KUKA KRL program: ap_2.src, ap_2.dat

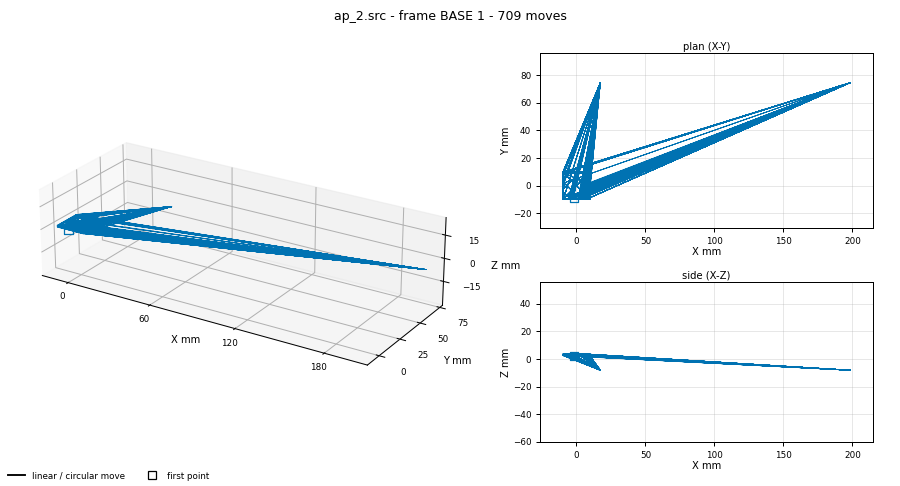
[picture p0: tool path of ap_2.src in frame BASE 1, 709 of 709 moves have a stored position in this frame; points joined in program order, loops and branches not executed]
--- ap_2.src ---
&ACCESS RVP
&REL 65
&PARAM DISKPATH = KRC:\R1\Program
DEF ap_2 ( )
   ;FOLD INI;%{PE}
     ;FOLD BASISTECH INI
       GLOBAL INTERRUPT DECL 3 WHEN $STOPMESS==TRUE DO IR_STOPM ( )
       INTERRUPT ON 3
       BAS (#INITMOV,0 )
     ;ENDFOLD (BASISTECH INI)
     ;FOLD USER INI
       ;Make your modifications here
     ;ENDFOLD (USER INI)
   ;ENDFOLD (INI)

   BAS (#VEL_PTP, 0020.0000)
   BAS (#ACC_PTP, 0020.0000)

   ;-----SET LIN AND ARC MOTION VARIABLES-----
   $VEL.ORI1 = 0350.0000
   $VEL.ORI2 = 0350.0000

   $ACC.CP = 0005.0000
   $ACC.ORI1 = 1000.0000
   $ACC.ORI2 = 1000.0000

   ;-----APPROXIMATION-----
   $APO.CVEL = 0100
   $APO.CPTP = 0100
   $APO.CDIS = 0006.0000
   $APO.CORI = 0090.0000

   BAS (#BASE, 1) ;Positioner
   BAS (#TOOL, 1) ;Vrashatel

   BAS(#VEL_PTP,15)                         ;;Set PTP Axis Velocity
   BAS(#ACC_PTP,50)                         ;;Set PTP Axis Acceleration
   PTP{A1 -92,A2 -133,A3 132,A4 7,A5 50,A6 -10}
   $VEL.CP = 0.060
   LIN  {X -1.968, Y -9.039, Z 2.300, A 0.000, B 0.000, C 0.000} C_DIS
   $VEL.CP = 0.060
   LIN  {X -5.102, Y -9.039, Z 2.300, A 0.000, B 0.000, C 0.000} C_DIS
   $VEL.CP = 0.060
   LIN  {X -9.039, Y -5.102, Z 2.300, A 0.000, B 0.000, C 0.000} C_DIS
   $VEL.CP = 0.060
   LIN  {X -9.039, Y -9.039, Z 2.300, A 0.000, B 0.000, C 0.000} C_DIS
   $VEL.CP = 0.060
   LIN  {X 9.039, Y 9.039, Z 2.300, A 0.000, B 0.000, C 0.000} C_DIS
   $VEL.CP = 0.060
   LIN  {X 9.040, Y 9.040, Z 2.300, A 0.000, B 0.000, C 0.000} C_DIS
   $VEL.CP = 0.060
   LIN  {X 9.039, Y 5.102, Z 2.300, A 0.000, B 0.000, C 0.000} C_DIS
   $VEL.CP = 0.060
   LIN  {X 5.102, Y 9.039, Z 2.300, A 0.000, B 0.000, C 0.000} C_DIS
   $VEL.CP = 0.060
   LIN  {X 1.968, Y 9.039, Z 2.300, A 0.000, B 0.000, C 0.000} C_DIS
   $VEL.CP = 0.060
   LIN  {X -9.039, Y -1.968, Z 2.300, A 0.000, B 0.000, C 0.000} C_DIS
   $VEL.CP = 0.060
   LIN  {X -9.039, Y 1.968, Z 2.300, A 0.000, B 0.000, C 0.000} C_DIS
   $VEL.CP = 0.060
   LIN  {X 1.968, Y -9.039, Z 2.300, A 0.000, B 0.000, C 0.000} C_DIS
   $VEL.CP = 0.060
   LIN  {X 9.040, Y -9.040, Z 2.300, A 0.000, B 0.000, C 0.000} C_DIS

;FOLD ARCOFF WDAT2 LIN P4 CPDAT2 Tool[1]:cmttorch Base[1]:vrashatel ;%{PE}
  ;FOLD Parameters ;%{h}
    ;Params IlfProvider=kukaroboter.arctech.arcofflin; Kuka.IsGlobalPoint=False; Kuka.PointName=P4; Kuka.BlendingEnabled=False; Kuka.MoveDataName=CPDAT2; Kuka.VelocityPath=0.01; Kuka.CurrentCDSetIndex=0; Kuka.MovementParameterFieldEnabled=True; ArcTech.WdatVarName=WDAT2; ArcTech.Basic=3.4.3.1264
  ;ENDFOLD
  $BWDSTART = FALSE
  LDAT_ACT = LCPDAT2
  FDAT_ACT = FP4
  BAS(#CP_PARAMS, gArcBasVelDefinition)
  SET_CD_PARAMS (0)
  TRIGGER WHEN PATH = ArcGetPath(#ArcOffBefore, WDAT2) DELAY = 0 DO ArcMainNG(#ArcOffBeforeOffStd, WDAT2, WP4) PRIO = -1
  TRIGGER WHEN PATH = ArcGetPath(#OnTheFlyArcOff, WDAT2) DELAY = 0 DO ArcMainNG(#ArcOffMoveStd, WDAT2, WP4) PRIO = -1
  ArcMainNG(#ArcOffBeforeMoveStd, WDAT2, WP4)
  LIN XP4
  ArcMainNG(#ArcOffAfterMoveStd, WDAT2, WP4)
;ENDFOLD
   $VEL.CP = 0.080
   LIN  {X 9.039, Y -9.039, Z 2.300, A 0.000, B 0.000, C 0.000} C_DIS

;FOLD ARCON WDAT1 LIN P3 Vel=0.5 m/s CPDAT1 Tool[1]:cmttorch Base[1]:vrashatel ;%{PE}
  ;FOLD Parameters ;%{h}
    ;Params IlfProvider=kukaroboter.arctech.arconlin; Kuka.IsGlobalPoint=False; Kuka.PointName=P3; Kuka.BlendingEnabled=False; Kuka.MoveDataName=CPDAT1; Kuka.VelocityPath=0.5; Kuka.CurrentCDSetIndex=0; Kuka.MovementParameterFieldEnabled=True; ArcTech.WdatVarName=WDAT1; ArcTech.Basic=3.4.3.1264
  ;ENDFOLD
  $BWDSTART = FALSE
  LDAT_ACT = LCPDAT1
  FDAT_ACT = FP3
  BAS(#CP_PARAMS, 0.5)
  SET_CD_PARAMS (0)
  TRIGGER WHEN DISTANCE = 1 DELAY = ArcGetDelay(#PreDefinition, WDAT1) DO ArcMainNG(#PreDefinition, WDAT1, WP3) PRIO = -1
  TRIGGER WHEN PATH = ArcGetPath(#OnTheFlyArcOn, WDAT1) DELAY = ArcGetDelay(#GasPreflow, WDAT1) DO ArcMainNG(#GasPreflow, WDAT1, WP3) PRIO = -1
  TRIGGER WHEN PATH = ArcGetPath(#OnTheFlyArcOn, WDAT1) DELAY = 0 DO ArcMainNG(#ArcOnMoveStd, WDAT1, WP3) PRIO = -1
  ArcMainNG(#ArcOnBeforeMoveStd, WDAT1, WP3)
  LIN XP3
  ArcMainNG(#ArcOnAfterMoveStd, WDAT1, WP3)
;ENDFOLD
   $VEL.CP = 0.060
   LIN  {X -9.039, Y 9.039, Z 2.300, A 0.000, B 0.000, C 0.000} C_DIS
   $VEL.CP = 0.060
   LIN  {X -9.040, Y 9.040, Z 2.300, A 0.000, B 0.000, C 0.000} C_DIS

;FOLD ARCOFF WDAT2 LIN P4 CPDAT2 Tool[1]:cmttorch Base[1]:vrashatel ;%{PE}
  ;FOLD Parameters ;%{h}
    ;Params IlfProvider=kukaroboter.arctech.arcofflin; Kuka.IsGlobalPoint=False; Kuka.PointName=P4; Kuka.BlendingEnabled=False; Kuka.MoveDataName=CPDAT2; Kuka.VelocityPath=0.01; Kuka.CurrentCDSetIndex=0; Kuka.MovementParameterFieldEnabled=True; ArcTech.WdatVarName=WDAT2; ArcTech.Basic=3.4.3.1264
  ;ENDFOLD
  $BWDSTART = FALSE
  LDAT_ACT = LCPDAT2
  FDAT_ACT = FP4
  BAS(#CP_PARAMS, gArcBasVelDefinition)
  SET_CD_PARAMS (0)
  TRIGGER WHEN PATH = ArcGetPath(#ArcOffBefore, WDAT2) DELAY = 0 DO ArcMainNG(#ArcOffBeforeOffStd, WDAT2, WP4) PRIO = -1
  TRIGGER WHEN PATH = ArcGetPath(#OnTheFlyArcOff, WDAT2) DELAY = 0 DO ArcMainNG(#ArcOffMoveStd, WDAT2, WP4) PRIO = -1
  ArcMainNG(#ArcOffBeforeMoveStd, WDAT2, WP4)
  LIN XP4
  ArcMainNG(#ArcOffAfterMoveStd, WDAT2, WP4)
;ENDFOLD
   $VEL.CP = 0.080
   LIN  {X 5.102, Y -9.039, Z 2.300, A 0.000, B 0.000, C 0.000} C_DIS

;FOLD ARCON WDAT1 LIN P3 Vel=0.5 m/s CPDAT1 Tool[1]:cmttorch Base[1]:vrashatel ;%{PE}
  ;FOLD Parameters ;%{h}
    ;Params IlfProvider=kukaroboter.arctech.arconlin; Kuka.IsGlobalPoint=False; Kuka.PointName=P3; Kuka.BlendingEnabled=False; Kuka.MoveDataName=CPDAT1; Kuka.VelocityPath=0.5; Kuka.CurrentCDSetIndex=0; Kuka.MovementParameterFieldEnabled=True; ArcTech.WdatVarName=WDAT1; ArcTech.Basic=3.4.3.1264
  ;ENDFOLD
  $BWDSTART = FALSE
  LDAT_ACT = LCPDAT1
  FDAT_ACT = FP3
  BAS(#CP_PARAMS, 0.5)
  SET_CD_PARAMS (0)
  TRIGGER WHEN DISTANCE = 1 DELAY = ArcGetDelay(#PreDefinition, WDAT1) DO ArcMainNG(#PreDefinition, WDAT1, WP3) PRIO = -1
  TRIGGER WHEN PATH = ArcGetPath(#OnTheFlyArcOn, WDAT1) DELAY = ArcGetDelay(#GasPreflow, WDAT1) DO ArcMainNG(#GasPreflow, WDAT1, WP3) PRIO = -1
  TRIGGER WHEN PATH = ArcGetPath(#OnTheFlyArcOn, WDAT1) DELAY = 0 DO ArcMainNG(#ArcOnMoveStd, WDAT1, WP3) PRIO = -1
  ArcMainNG(#ArcOnBeforeMoveStd, WDAT1, WP3)
  LIN XP3
  ArcMainNG(#ArcOnAfterMoveStd, WDAT1, WP3)
;ENDFOLD
   $VEL.CP = 0.025
   LIN  {X 5.102, Y -9.039, Z 2.300, A 0.000, B 0.000, C 0.000} C_DIS
   $VEL.CP = 0.060
   LIN  {X 9.039, Y -5.102, Z 2.300, A 0.000, B 0.000, C 0.000} C_DIS
   $VEL.CP = 0.060
   LIN  {X 9.039, Y -9.039, Z 2.300, A 0.000, B 0.000, C 0.000} C_DIS

;FOLD ARCOFF WDAT2 LIN P4 CPDAT2 Tool[1]:cmttorch Base[1]:vrashatel ;%{PE}
  ;FOLD Parameters ;%{h}
    ;Params IlfProvider=kukaroboter.arctech.arcofflin; Kuka.IsGlobalPoint=False; Kuka.PointName=P4; Kuka.BlendingEnabled=False; Kuka.MoveDataName=CPDAT2; Kuka.VelocityPath=0.01; Kuka.CurrentCDSetIndex=0; Kuka.MovementParameterFieldEnabled=True; ArcTech.WdatVarName=WDAT2; ArcTech.Basic=3.4.3.1264
  ;ENDFOLD
  $BWDSTART = FALSE
  LDAT_ACT = LCPDAT2
  FDAT_ACT = FP4
  BAS(#CP_PARAMS, gArcBasVelDefinition)
  SET_CD_PARAMS (0)
  TRIGGER WHEN PATH = ArcGetPath(#ArcOffBefore, WDAT2) DELAY = 0 DO ArcMainNG(#ArcOffBeforeOffStd, WDAT2, WP4) PRIO = -1
  TRIGGER WHEN PATH = ArcGetPath(#OnTheFlyArcOff, WDAT2) DELAY = 0 DO ArcMainNG(#ArcOffMoveStd, WDAT2, WP4) PRIO = -1
  ArcMainNG(#ArcOffBeforeMoveStd, WDAT2, WP4)
  LIN XP4
  ArcMainNG(#ArcOffAfterMoveStd, WDAT2, WP4)
;ENDFOLD
   $VEL.CP = 0.060
   LIN  {X 9.039, Y -9.139, Z 2.300, A 0.000, B 0.000, C 0.000} C_DIS
   $VEL.CP = 0.010
   LIN  {X 9.039, Y -9.139, Z 2.500, A 0.000, B 0.000, C 0.000} C_DIS
   $VEL.CP = 0.080
   LIN  {X -9.530, Y 9.530, Z 2.500, A 0.000, B 0.000, C 0.000} C_DIS
   $VEL.CP = 0.080
   LIN  {X -9.800, Y 9.800, Z 2.500, A 0.000, B 0.000, C 0.000} C_DIS

;FOLD ARCON WDAT1 LIN P3 Vel=0.5 m/s CPDAT1 Tool[1]:cmttorch Base[1]:vrashatel ;%{PE}
  ;FOLD Parameters ;%{h}
    ;Params IlfProvider=kukaroboter.arctech.arconlin; Kuka.IsGlobalPoint=False; Kuka.PointName=P3; Kuka.BlendingEnabled=False; Kuka.MoveDataName=CPDAT1; Kuka.VelocityPath=0.5; Kuka.CurrentCDSetIndex=0; Kuka.MovementParameterFieldEnabled=True; ArcTech.WdatVarName=WDAT1; ArcTech.Basic=3.4.3.1264
  ;ENDFOLD
  $BWDSTART = FALSE
  LDAT_ACT = LCPDAT1
  FDAT_ACT = FP3
  BAS(#CP_PARAMS, 0.5)
  SET_CD_PARAMS (0)
  TRIGGER WHEN DISTANCE = 1 DELAY = ArcGetDelay(#PreDefinition, WDAT1) DO ArcMainNG(#PreDefinition, WDAT1, WP3) PRIO = -1
  TRIGGER WHEN PATH = ArcGetPath(#OnTheFlyArcOn, WDAT1) DELAY = ArcGetDelay(#GasPreflow, WDAT1) DO ArcMainNG(#GasPreflow, WDAT1, WP3) PRIO = -1
  TRIGGER WHEN PATH = ArcGetPath(#OnTheFlyArcOn, WDAT1) DELAY = 0 DO ArcMainNG(#ArcOnMoveStd, WDAT1, WP3) PRIO = -1
  ArcMainNG(#ArcOnBeforeMoveStd, WDAT1, WP3)
  LIN XP3
  ArcMainNG(#ArcOnAfterMoveStd, WDAT1, WP3)
;ENDFOLD
   $VEL.CP = 0.025
   LIN  {X -9.800, Y 9.800, Z 2.500, A 0.000, B 0.000, C 0.000} C_DIS
   $VEL.CP = 0.060
   LIN  {X -9.800, Y -9.800, Z 2.500, A 0.000, B 0.000, C 0.000} C_DIS
   $VEL.CP = 0.060
   LIN  {X 9.800, Y -9.800, Z 2.500, A 0.000, B 0.000, C 0.000} C_DIS
   $VEL.CP = 0.060
   LIN  {X 9.800, Y 9.800, Z 2.500, A 0.000, B 0.000, C 0.000} C_DIS
   $VEL.CP = 0.060
   LIN  {X -9.800, Y 9.800, Z 2.500, A 0.000, B 0.000, C 0.000} C_DIS

;FOLD ARCOFF WDAT2 LIN P4 CPDAT2 Tool[1]:cmttorch Base[1]:vrashatel ;%{PE}
  ;FOLD Parameters ;%{h}
    ;Params IlfProvider=kukaroboter.arctech.arcofflin; Kuka.IsGlobalPoint=False; Kuka.PointName=P4; Kuka.BlendingEnabled=False; Kuka.MoveDataName=CPDAT2; Kuka.VelocityPath=0.01; Kuka.CurrentCDSetIndex=0; Kuka.MovementParameterFieldEnabled=True; ArcTech.WdatVarName=WDAT2; ArcTech.Basic=3.4.3.1264
  ;ENDFOLD
  $BWDSTART = FALSE
  LDAT_ACT = LCPDAT2
  FDAT_ACT = FP4
  BAS(#CP_PARAMS, gArcBasVelDefinition)
  SET_CD_PARAMS (0)
  TRIGGER WHEN PATH = ArcGetPath(#ArcOffBefore, WDAT2) DELAY = 0 DO ArcMainNG(#ArcOffBeforeOffStd, WDAT2, WP4) PRIO = -1
  TRIGGER WHEN PATH = ArcGetPath(#OnTheFlyArcOff, WDAT2) DELAY = 0 DO ArcMainNG(#ArcOffMoveStd, WDAT2, WP4) PRIO = -1
  ArcMainNG(#ArcOffBeforeMoveStd, WDAT2, WP4)
  LIN XP4
  ArcMainNG(#ArcOffAfterMoveStd, WDAT2, WP4)
;ENDFOLD
   $VEL.CP = 0.080
   LIN  {X -9.800, Y 9.600, Z 2.500, A 0.000, B 0.000, C 0.000} C_DIS
   $VEL.CP = 0.080
   LIN  {X -9.360, Y 9.360, Z 2.500, A 0.000, B 0.000, C 0.000} C_DIS
   $VEL.CP = 0.080
   LIN  {X -9.400, Y 9.400, Z 2.500, A 0.000, B 0.000, C 0.000} C_DIS

;FOLD ARCON WDAT1 LIN P3 Vel=0.5 m/s CPDAT1 Tool[1]:cmttorch Base[1]:vrashatel ;%{PE}
  ;FOLD Parameters ;%{h}
    ;Params IlfProvider=kukaroboter.arctech.arconlin; Kuka.IsGlobalPoint=False; Kuka.PointName=P3; Kuka.BlendingEnabled=False; Kuka.MoveDataName=CPDAT1; Kuka.VelocityPath=0.5; Kuka.CurrentCDSetIndex=0; Kuka.MovementParameterFieldEnabled=True; ArcTech.WdatVarName=WDAT1; ArcTech.Basic=3.4.3.1264
  ;ENDFOLD
  $BWDSTART = FALSE
  LDAT_ACT = LCPDAT1
  FDAT_ACT = FP3
  BAS(#CP_PARAMS, 0.5)
  SET_CD_PARAMS (0)
  TRIGGER WHEN DISTANCE = 1 DELAY = ArcGetDelay(#PreDefinition, WDAT1) DO ArcMainNG(#PreDefinition, WDAT1, WP3) PRIO = -1
  TRIGGER WHEN PATH = ArcGetPath(#OnTheFlyArcOn, WDAT1) DELAY = ArcGetDelay(#GasPreflow, WDAT1) DO ArcMainNG(#GasPreflow, WDAT1, WP3) PRIO = -1
  TRIGGER WHEN PATH = ArcGetPath(#OnTheFlyArcOn, WDAT1) DELAY = 0 DO ArcMainNG(#ArcOnMoveStd, WDAT1, WP3) PRIO = -1
  ArcMainNG(#ArcOnBeforeMoveStd, WDAT1, WP3)
  LIN XP3
  ArcMainNG(#ArcOnAfterMoveStd, WDAT1, WP3)
;ENDFOLD
   $VEL.CP = 0.060
   LIN  {X -9.400, Y -9.400, Z 2.500, A 0.000, B 0.000, C 0.000} C_DIS
   $VEL.CP = 0.060
   LIN  {X 9.400, Y -9.400, Z 2.500, A 0.000, B 0.000, C 0.000} C_DIS
   $VEL.CP = 0.060
   LIN  {X 9.400, Y 9.400, Z 2.500, A 0.000, B 0.000, C 0.000} C_DIS
   $VEL.CP = 0.060
   LIN  {X -9.400, Y 9.400, Z 2.500, A 0.000, B 0.000, C 0.000} C_DIS

;FOLD ARCOFF WDAT2 LIN P4 CPDAT2 Tool[1]:cmttorch Base[1]:vrashatel ;%{PE}
  ;FOLD Parameters ;%{h}
    ;Params IlfProvider=kukaroboter.arctech.arcofflin; Kuka.IsGlobalPoint=False; Kuka.PointName=P4; Kuka.BlendingEnabled=False; Kuka.MoveDataName=CPDAT2; Kuka.VelocityPath=0.01; Kuka.CurrentCDSetIndex=0; Kuka.MovementParameterFieldEnabled=True; ArcTech.WdatVarName=WDAT2; ArcTech.Basic=3.4.3.1264
  ;ENDFOLD
  $BWDSTART = FALSE
  LDAT_ACT = LCPDAT2
  FDAT_ACT = FP4
  BAS(#CP_PARAMS, gArcBasVelDefinition)
  SET_CD_PARAMS (0)
  TRIGGER WHEN PATH = ArcGetPath(#ArcOffBefore, WDAT2) DELAY = 0 DO ArcMainNG(#ArcOffBeforeOffStd, WDAT2, WP4) PRIO = -1
  TRIGGER WHEN PATH = ArcGetPath(#OnTheFlyArcOff, WDAT2) DELAY = 0 DO ArcMainNG(#ArcOffMoveStd, WDAT2, WP4) PRIO = -1
  ArcMainNG(#ArcOffBeforeMoveStd, WDAT2, WP4)
  LIN XP4
  ArcMainNG(#ArcOffAfterMoveStd, WDAT2, WP4)
;ENDFOLD
   $VEL.CP = 0.080
   LIN  {X -9.040, Y 9.040, Z 2.500, A 0.000, B 0.000, C 0.000} C_DIS

;FOLD ARCON WDAT1 LIN P3 Vel=0.5 m/s CPDAT1 Tool[1]:cmttorch Base[1]:vrashatel ;%{PE}
  ;FOLD Parameters ;%{h}
    ;Params IlfProvider=kukaroboter.arctech.arconlin; Kuka.IsGlobalPoint=False; Kuka.PointName=P3; Kuka.BlendingEnabled=False; Kuka.MoveDataName=CPDAT1; Kuka.VelocityPath=0.5; Kuka.CurrentCDSetIndex=0; Kuka.MovementParameterFieldEnabled=True; ArcTech.WdatVarName=WDAT1; ArcTech.Basic=3.4.3.1264
  ;ENDFOLD
  $BWDSTART = FALSE
  LDAT_ACT = LCPDAT1
  FDAT_ACT = FP3
  BAS(#CP_PARAMS, 0.5)
  SET_CD_PARAMS (0)
  TRIGGER WHEN DISTANCE = 1 DELAY = ArcGetDelay(#PreDefinition, WDAT1) DO ArcMainNG(#PreDefinition, WDAT1, WP3) PRIO = -1
  TRIGGER WHEN PATH = ArcGetPath(#OnTheFlyArcOn, WDAT1) DELAY = ArcGetDelay(#GasPreflow, WDAT1) DO ArcMainNG(#GasPreflow, WDAT1, WP3) PRIO = -1
  TRIGGER WHEN PATH = ArcGetPath(#OnTheFlyArcOn, WDAT1) DELAY = 0 DO ArcMainNG(#ArcOnMoveStd, WDAT1, WP3) PRIO = -1
  ArcMainNG(#ArcOnBeforeMoveStd, WDAT1, WP3)
  LIN XP3
  ArcMainNG(#ArcOnAfterMoveStd, WDAT1, WP3)
;ENDFOLD
   $VEL.CP = 0.060
   LIN  {X -9.039, Y 5.102, Z 2.500, A 0.000, B 0.000, C 0.000} C_DIS
   $VEL.CP = 0.060
   LIN  {X -5.102, Y 9.039, Z 2.500, A 0.000, B 0.000, C 0.000} C_DIS
   $VEL.CP = 0.060
   LIN  {X -1.968, Y 9.039, Z 2.500, A 0.000, B 0.000, C 0.000} C_DIS
   $VEL.CP = 0.060
   LIN  {X 9.039, Y -1.968, Z 2.500, A 0.000, B 0.000, C 0.000} C_DIS
   $VEL.CP = 0.060
   LIN  {X 9.039, Y 1.968, Z 2.500, A 0.000, B 0.000, C 0.000} C_DIS
   $VEL.CP = 0.060
   LIN  {X -1.968, Y -9.039, Z 2.500, A 0.000, B 0.000, C 0.000} C_DIS
   $VEL.CP = 0.060
   LIN  {X -5.102, Y -9.039, Z 2.500, A 0.000, B 0.000, C 0.000} C_DIS
   $VEL.CP = 0.060
   LIN  {X -9.039, Y -5.102, Z 2.500, A 0.000, B 0.000, C 0.000} C_DIS
   $VEL.CP = 0.060
   LIN  {X -9.039, Y -9.039, Z 2.500, A 0.000, B 0.000, C 0.000} C_DIS
   $VEL.CP = 0.060
   LIN  {X 9.039, Y 9.039, Z 2.500, A 0.000, B 0.000, C 0.000} C_DIS
   $VEL.CP = 0.060
   LIN  {X 9.040, Y 9.040, Z 2.500, A 0.000, B 0.000, C 0.000} C_DIS
   $VEL.CP = 0.060
   LIN  {X 9.039, Y 5.102, Z 2.500, A 0.000, B 0.000, C 0.000} C_DIS
   $VEL.CP = 0.060
   LIN  {X 5.102, Y 9.039, Z 2.500, A 0.000, B 0.000, C 0.000} C_DIS
   $VEL.CP = 0.060
   LIN  {X 1.968, Y 9.039, Z 2.500, A 0.000, B 0.000, C 0.000} C_DIS
   $VEL.CP = 0.060
   LIN  {X -9.039, Y -1.968, Z 2.500, A 0.000, B 0.000, C 0.000} C_DIS
   $VEL.CP = 0.060
   LIN  {X -9.039, Y 1.968, Z 2.500, A 0.000, B 0.000, C 0.000} C_DIS
   $VEL.CP = 0.060
   LIN  {X 1.968, Y -9.039, Z 2.500, A 0.000, B 0.000, C 0.000} C_DIS
   $VEL.CP = 0.060
   LIN  {X 9.040, Y -9.040, Z 2.500, A 0.000, B 0.000, C 0.000} C_DIS

;FOLD ARCOFF WDAT2 LIN P4 CPDAT2 Tool[1]:cmttorch Base[1]:vrashatel ;%{PE}
  ;FOLD Parameters ;%{h}
    ;Params IlfProvider=kukaroboter.arctech.arcofflin; Kuka.IsGlobalPoint=False; Kuka.PointName=P4; Kuka.BlendingEnabled=False; Kuka.MoveDataName=CPDAT2; Kuka.VelocityPath=0.01; Kuka.CurrentCDSetIndex=0; Kuka.MovementParameterFieldEnabled=True; ArcTech.WdatVarName=WDAT2; ArcTech.Basic=3.4.3.1264
  ;ENDFOLD
  $BWDSTART = FALSE
  LDAT_ACT = LCPDAT2
  FDAT_ACT = FP4
  BAS(#CP_PARAMS, gArcBasVelDefinition)
  SET_CD_PARAMS (0)
  TRIGGER WHEN PATH = ArcGetPath(#ArcOffBefore, WDAT2) DELAY = 0 DO ArcMainNG(#ArcOffBeforeOffStd, WDAT2, WP4) PRIO = -1
  TRIGGER WHEN PATH = ArcGetPath(#OnTheFlyArcOff, WDAT2) DELAY = 0 DO ArcMainNG(#ArcOffMoveStd, WDAT2, WP4) PRIO = -1
  ArcMainNG(#ArcOffBeforeMoveStd, WDAT2, WP4)
  LIN XP4
  ArcMainNG(#ArcOffAfterMoveStd, WDAT2, WP4)
;ENDFOLD
   $VEL.CP = 0.080
   LIN  {X 9.039, Y -9.039, Z 2.500, A 0.000, B 0.000, C 0.000} C_DIS

;FOLD ARCON WDAT1 LIN P3 Vel=0.5 m/s CPDAT1 Tool[1]:cmttorch Base[1]:vrashatel ;%{PE}
  ;FOLD Parameters ;%{h}
    ;Params IlfProvider=kukaroboter.arctech.arconlin; Kuka.IsGlobalPoint=False; Kuka.PointName=P3; Kuka.BlendingEnabled=False; Kuka.MoveDataName=CPDAT1; Kuka.VelocityPath=0.5; Kuka.CurrentCDSetIndex=0; Kuka.MovementParameterFieldEnabled=True; ArcTech.WdatVarName=WDAT1; ArcTech.Basic=3.4.3.1264
  ;ENDFOLD
  $BWDSTART = FALSE
  LDAT_ACT = LCPDAT1
  FDAT_ACT = FP3
  BAS(#CP_PARAMS, 0.5)
  SET_CD_PARAMS (0)
  TRIGGER WHEN DISTANCE = 1 DELAY = ArcGetDelay(#PreDefinition, WDAT1) DO ArcMainNG(#PreDefinition, WDAT1, WP3) PRIO = -1
  TRIGGER WHEN PATH = ArcGetPath(#OnTheFlyArcOn, WDAT1) DELAY = ArcGetDelay(#GasPreflow, WDAT1) DO ArcMainNG(#GasPreflow, WDAT1, WP3) PRIO = -1
  TRIGGER WHEN PATH = ArcGetPath(#OnTheFlyArcOn, WDAT1) DELAY = 0 DO ArcMainNG(#ArcOnMoveStd, WDAT1, WP3) PRIO = -1
  ArcMainNG(#ArcOnBeforeMoveStd, WDAT1, WP3)
  LIN XP3
  ArcMainNG(#ArcOnAfterMoveStd, WDAT1, WP3)
;ENDFOLD
   $VEL.CP = 0.060
   LIN  {X -9.039, Y 9.039, Z 2.500, A 0.000, B 0.000, C 0.000} C_DIS
   $VEL.CP = 0.060
   LIN  {X -9.040, Y 9.040, Z 2.500, A 0.000, B 0.000, C 0.000} C_DIS

;FOLD ARCOFF WDAT2 LIN P4 CPDAT2 Tool[1]:cmttorch Base[1]:vrashatel ;%{PE}
  ;FOLD Parameters ;%{h}
    ;Params IlfProvider=kukaroboter.arctech.arcofflin; Kuka.IsGlobalPoint=False; Kuka.PointName=P4; Kuka.BlendingEnabled=False; Kuka.MoveDataName=CPDAT2; Kuka.VelocityPath=0.01; Kuka.CurrentCDSetIndex=0; Kuka.MovementParameterFieldEnabled=True; ArcTech.WdatVarName=WDAT2; ArcTech.Basic=3.4.3.1264
  ;ENDFOLD
  $BWDSTART = FALSE
  LDAT_ACT = LCPDAT2
  FDAT_ACT = FP4
  BAS(#CP_PARAMS, gArcBasVelDefinition)
  SET_CD_PARAMS (0)
  TRIGGER WHEN PATH = ArcGetPath(#ArcOffBefore, WDAT2) DELAY = 0 DO ArcMainNG(#ArcOffBeforeOffStd, WDAT2, WP4) PRIO = -1
  TRIGGER WHEN PATH = ArcGetPath(#OnTheFlyArcOff, WDAT2) DELAY = 0 DO ArcMainNG(#ArcOffMoveStd, WDAT2, WP4) PRIO = -1
  ArcMainNG(#ArcOffBeforeMoveStd, WDAT2, WP4)
  LIN XP4
  ArcMainNG(#ArcOffAfterMoveStd, WDAT2, WP4)
;ENDFOLD
   $VEL.CP = 0.080
   LIN  {X 5.102, Y -9.039, Z 2.500, A 0.000, B 0.000, C 0.000} C_DIS

;FOLD ARCON WDAT1 LIN P3 Vel=0.5 m/s CPDAT1 Tool[1]:cmttorch Base[1]:vrashatel ;%{PE}
  ;FOLD Parameters ;%{h}
    ;Params IlfProvider=kukaroboter.arctech.arconlin; Kuka.IsGlobalPoint=False; Kuka.PointName=P3; Kuka.BlendingEnabled=False; Kuka.MoveDataName=CPDAT1; Kuka.VelocityPath=0.5; Kuka.CurrentCDSetIndex=0; Kuka.MovementParameterFieldEnabled=True; ArcTech.WdatVarName=WDAT1; ArcTech.Basic=3.4.3.1264
  ;ENDFOLD
  $BWDSTART = FALSE
  LDAT_ACT = LCPDAT1
  FDAT_ACT = FP3
  BAS(#CP_PARAMS, 0.5)
  SET_CD_PARAMS (0)
  TRIGGER WHEN DISTANCE = 1 DELAY = ArcGetDelay(#PreDefinition, WDAT1) DO ArcMainNG(#PreDefinition, WDAT1, WP3) PRIO = -1
  TRIGGER WHEN PATH = ArcGetPath(#OnTheFlyArcOn, WDAT1) DELAY = ArcGetDelay(#GasPreflow, WDAT1) DO ArcMainNG(#GasPreflow, WDAT1, WP3) PRIO = -1
  TRIGGER WHEN PATH = ArcGetPath(#OnTheFlyArcOn, WDAT1) DELAY = 0 DO ArcMainNG(#ArcOnMoveStd, WDAT1, WP3) PRIO = -1
  ArcMainNG(#ArcOnBeforeMoveStd, WDAT1, WP3)
  LIN XP3
  ArcMainNG(#ArcOnAfterMoveStd, WDAT1, WP3)
;ENDFOLD
   $VEL.CP = 0.025
   LIN  {X 5.102, Y -9.039, Z 2.500, A 0.000, B 0.000, C 0.000} C_DIS
   $VEL.CP = 0.060
   LIN  {X 9.039, Y -5.102, Z 2.500, A 0.000, B 0.000, C 0.000} C_DIS
   $VEL.CP = 0.060
   LIN  {X 9.039, Y -9.039, Z 2.500, A 0.000, B 0.000, C 0.000} C_DIS

;FOLD ARCOFF WDAT2 LIN P4 CPDAT2 Tool[1]:cmttorch Base[1]:vrashatel ;%{PE}
  ;FOLD Parameters ;%{h}
    ;Params IlfProvider=kukaroboter.arctech.arcofflin; Kuka.IsGlobalPoint=False; Kuka.PointName=P4; Kuka.BlendingEnabled=False; Kuka.MoveDataName=CPDAT2; Kuka.VelocityPath=0.01; Kuka.CurrentCDSetIndex=0; Kuka.MovementParameterFieldEnabled=True; ArcTech.WdatVarName=WDAT2; ArcTech.Basic=3.4.3.1264
  ;ENDFOLD
  $BWDSTART = FALSE
  LDAT_ACT = LCPDAT2
  FDAT_ACT = FP4
  BAS(#CP_PARAMS, gArcBasVelDefinition)
  SET_CD_PARAMS (0)
  TRIGGER WHEN PATH = ArcGetPath(#ArcOffBefore, WDAT2) DELAY = 0 DO ArcMainNG(#ArcOffBeforeOffStd, WDAT2, WP4) PRIO = -1
  TRIGGER WHEN PATH = ArcGetPath(#OnTheFlyArcOff, WDAT2) DELAY = 0 DO ArcMainNG(#ArcOffMoveStd, WDAT2, WP4) PRIO = -1
  ArcMainNG(#ArcOffBeforeMoveStd, WDAT2, WP4)
  LIN XP4
  ArcMainNG(#ArcOffAfterMoveStd, WDAT2, WP4)
;ENDFOLD
   $VEL.CP = 0.060
   LIN  {X 9.039, Y -9.139, Z 2.500, A 0.000, B 0.000, C 0.000} C_DIS
   $VEL.CP = 0.010
   LIN  {X 9.039, Y -9.139, Z 2.700, A 0.000, B 0.000, C 0.000} C_DIS
   $VEL.CP = 0.080
   LIN  {X -9.530, Y 9.530, Z 2.700, A 0.000, B 0.000, C 0.000} C_DIS
   $VEL.CP = 0.080
   LIN  {X -9.800, Y 9.800, Z 2.700, A 0.000, B 0.000, C 0.000} C_DIS

;FOLD ARCON WDAT1 LIN P3 Vel=0.5 m/s CPDAT1 Tool[1]:cmttorch Base[1]:vrashatel ;%{PE}
  ;FOLD Parameters ;%{h}
    ;Params IlfProvider=kukaroboter.arctech.arconlin; Kuka.IsGlobalPoint=False; Kuka.PointName=P3; Kuka.BlendingEnabled=False; Kuka.MoveDataName=CPDAT1; Kuka.VelocityPath=0.5; Kuka.CurrentCDSetIndex=0; Kuka.MovementParameterFieldEnabled=True; ArcTech.WdatVarName=WDAT1; ArcTech.Basic=3.4.3.1264
  ;ENDFOLD
  $BWDSTART = FALSE
  LDAT_ACT = LCPDAT1
  FDAT_ACT = FP3
  BAS(#CP_PARAMS, 0.5)
  SET_CD_PARAMS (0)
  TRIGGER WHEN DISTANCE = 1 DELAY = ArcGetDelay(#PreDefinition, WDAT1) DO ArcMainNG(#PreDefinition, WDAT1, WP3) PRIO = -1
  TRIGGER WHEN PATH = ArcGetPath(#OnTheFlyArcOn, WDAT1) DELAY = ArcGetDelay(#GasPreflow, WDAT1) DO ArcMainNG(#GasPreflow, WDAT1, WP3) PRIO = -1
  TRIGGER WHEN PATH = ArcGetPath(#OnTheFlyArcOn, WDAT1) DELAY = 0 DO ArcMainNG(#ArcOnMoveStd, WDAT1, WP3) PRIO = -1
  ArcMainNG(#ArcOnBeforeMoveStd, WDAT1, WP3)
  LIN XP3
  ArcMainNG(#ArcOnAfterMoveStd, WDAT1, WP3)
;ENDFOLD
   $VEL.CP = 0.025
   LIN  {X -9.800, Y 9.800, Z 2.700, A 0.000, B 0.000, C 0.000} C_DIS
   $VEL.CP = 0.060
   LIN  {X -9.800, Y -9.800, Z 2.700, A 0.000, B 0.000, C 0.000} C_DIS
   $VEL.CP = 0.060
   LIN  {X 9.800, Y -9.800, Z 2.700, A 0.000, B 0.000, C 0.000} C_DIS
   $VEL.CP = 0.060
   LIN  {X 9.800, Y 9.800, Z 2.700, A 0.000, B 0.000, C 0.000} C_DIS
   $VEL.CP = 0.060
   LIN  {X -9.800, Y 9.800, Z 2.700, A 0.000, B 0.000, C 0.000} C_DIS

;FOLD ARCOFF WDAT2 LIN P4 CPDAT2 Tool[1]:cmttorch Base[1]:vrashatel ;%{PE}
  ;FOLD Parameters ;%{h}
    ;Params IlfProvider=kukaroboter.arctech.arcofflin; Kuka.IsGlobalPoint=False; Kuka.PointName=P4; Kuka.BlendingEnabled=False; Kuka.MoveDataName=CPDAT2; Kuka.VelocityPath=0.01; Kuka.CurrentCDSetIndex=0; Kuka.MovementParameterFieldEnabled=True; ArcTech.WdatVarName=WDAT2; ArcTech.Basic=3.4.3.1264
  ;ENDFOLD
  $BWDSTART = FALSE
  LDAT_ACT = LCPDAT2
  FDAT_ACT = FP4
  BAS(#CP_PARAMS, gArcBasVelDefinition)
  SET_CD_PARAMS (0)
  TRIGGER WHEN PATH = ArcGetPath(#ArcOffBefore, WDAT2) DELAY = 0 DO ArcMainNG(#ArcOffBeforeOffStd, WDAT2, WP4) PRIO = -1
  TRIGGER WHEN PATH = ArcGetPath(#OnTheFlyArcOff, WDAT2) DELAY = 0 DO ArcMainNG(#ArcOffMoveStd, WDAT2, WP4) PRIO = -1
  ArcMainNG(#ArcOffBeforeMoveStd, WDAT2, WP4)
  LIN XP4
  ArcMainNG(#ArcOffAfterMoveStd, WDAT2, WP4)
;ENDFOLD
   $VEL.CP = 0.080
   LIN  {X -9.800, Y 9.600, Z 2.700, A 0.000, B 0.000, C 0.000} C_DIS
   $VEL.CP = 0.080
   LIN  {X -9.360, Y 9.360, Z 2.700, A 0.000, B 0.000, C 0.000} C_DIS
   $VEL.CP = 0.080
   LIN  {X -9.400, Y 9.400, Z 2.700, A 0.000, B 0.000, C 0.000} C_DIS

;FOLD ARCON WDAT1 LIN P3 Vel=0.5 m/s CPDAT1 Tool[1]:cmttorch Base[1]:vrashatel ;%{PE}
  ;FOLD Parameters ;%{h}
    ;Params IlfProvider=kukaroboter.arctech.arconlin; Kuka.IsGlobalPoint=False; Kuka.PointName=P3; Kuka.BlendingEnabled=False; Kuka.MoveDataName=CPDAT1; Kuka.VelocityPath=0.5; Kuka.CurrentCDSetIndex=0; Kuka.MovementParameterFieldEnabled=True; ArcTech.WdatVarName=WDAT1; ArcTech.Basic=3.4.3.1264
  ;ENDFOLD
  $BWDSTART = FALSE
  LDAT_ACT = LCPDAT1
  FDAT_ACT = FP3
  BAS(#CP_PARAMS, 0.5)
  SET_CD_PARAMS (0)
  TRIGGER WHEN DISTANCE = 1 DELAY = ArcGetDelay(#PreDefinition, WDAT1) DO ArcMainNG(#PreDefinition, WDAT1, WP3) PRIO = -1
  TRIGGER WHEN PATH = ArcGetPath(#OnTheFlyArcOn, WDAT1) DELAY = ArcGetDelay(#GasPreflow, WDAT1) DO ArcMainNG(#GasPreflow, WDAT1, WP3) PRIO = -1
  TRIGGER WHEN PATH = ArcGetPath(#OnTheFlyArcOn, WDAT1) DELAY = 0 DO ArcMainNG(#ArcOnMoveStd, WDAT1, WP3) PRIO = -1
  ArcMainNG(#ArcOnBeforeMoveStd, WDAT1, WP3)
  LIN XP3
  ArcMainNG(#ArcOnAfterMoveStd, WDAT1, WP3)
;ENDFOLD
   $VEL.CP = 0.060
   LIN  {X -9.400, Y -9.400, Z 2.700, A 0.000, B 0.000, C 0.000} C_DIS
   $VEL.CP = 0.060
   LIN  {X 9.400, Y -9.400, Z 2.700, A 0.000, B 0.000, C 0.000} C_DIS
   $VEL.CP = 0.060
   LIN  {X 9.400, Y 9.400, Z 2.700, A 0.000, B 0.000, C 0.000} C_DIS
   $VEL.CP = 0.060
   LIN  {X -9.400, Y 9.400, Z 2.700, A 0.000, B 0.000, C 0.000} C_DIS

;FOLD ARCOFF WDAT2 LIN P4 CPDAT2 Tool[1]:cmttorch Base[1]:vrashatel ;%{PE}
  ;FOLD Parameters ;%{h}
    ;Params IlfProvider=kukaroboter.arctech.arcofflin; Kuka.IsGlobalPoint=False; Kuka.PointName=P4; Kuka.BlendingEnabled=False; Kuka.MoveDataName=CPDAT2; Kuka.VelocityPath=0.01; Kuka.CurrentCDSetIndex=0; Kuka.MovementParameterFieldEnabled=True; ArcTech.WdatVarName=WDAT2; ArcTech.Basic=3.4.3.1264
  ;ENDFOLD
  $BWDSTART = FALSE
  LDAT_ACT = LCPDAT2
  FDAT_ACT = FP4
  BAS(#CP_PARAMS, gArcBasVelDefinition)
  SET_CD_PARAMS (0)
  TRIGGER WHEN PATH = ArcGetPath(#ArcOffBefore, WDAT2) DELAY = 0 DO ArcMainNG(#ArcOffBeforeOffStd, WDAT2, WP4) PRIO = -1
  TRIGGER WHEN PATH = ArcGetPath(#OnTheFlyArcOff, WDAT2) DELAY = 0 DO ArcMainNG(#ArcOffMoveStd, WDAT2, WP4) PRIO = -1
  ArcMainNG(#ArcOffBeforeMoveStd, WDAT2, WP4)
  LIN XP4
  ArcMainNG(#ArcOffAfterMoveStd, WDAT2, WP4)
;ENDFOLD
   $VEL.CP = 0.080
   LIN  {X -9.040, Y 9.040, Z 2.700, A 0.000, B 0.000, C 0.000} C_DIS

;FOLD ARCON WDAT1 LIN P3 Vel=0.5 m/s CPDAT1 Tool[1]:cmttorch Base[1]:vrashatel ;%{PE}
  ;FOLD Parameters ;%{h}
    ;Params IlfProvider=kukaroboter.arctech.arconlin; Kuka.IsGlobalPoint=False; Kuka.PointName=P3; Kuka.BlendingEnabled=False; Kuka.MoveDataName=CPDAT1; Kuka.VelocityPath=0.5; Kuka.CurrentCDSetIndex=0; Kuka.MovementParameterFieldEnabled=True; ArcTech.WdatVarName=WDAT1; ArcTech.Basic=3.4.3.1264
  ;ENDFOLD
  $BWDSTART = FALSE
  LDAT_ACT = LCPDAT1
  FDAT_ACT = FP3
  BAS(#CP_PARAMS, 0.5)
  SET_CD_PARAMS (0)
  TRIGGER WHEN DISTANCE = 1 DELAY = ArcGetDelay(#PreDefinition, WDAT1) DO ArcMainNG(#PreDefinition, WDAT1, WP3) PRIO = -1
  TRIGGER WHEN PATH = ArcGetPath(#OnTheFlyArcOn, WDAT1) DELAY = ArcGetDelay(#GasPreflow, WDAT1) DO ArcMainNG(#GasPreflow, WDAT1, WP3) PRIO = -1
  TRIGGER WHEN PATH = ArcGetPath(#OnTheFlyArcOn, WDAT1) DELAY = 0 DO ArcMainNG(#ArcOnMoveStd, WDAT1, WP3) PRIO = -1
  ArcMainNG(#ArcOnBeforeMoveStd, WDAT1, WP3)
  LIN XP3
  ArcMainNG(#ArcOnAfterMoveStd, WDAT1, WP3)
;ENDFOLD
   $VEL.CP = 0.060
   LIN  {X -9.039, Y 5.102, Z 2.700, A 0.000, B 0.000, C 0.000} C_DIS
   $VEL.CP = 0.060
   LIN  {X -5.102, Y 9.039, Z 2.700, A 0.000, B 0.000, C 0.000} C_DIS
   $VEL.CP = 0.060
   LIN  {X -1.968, Y 9.039, Z 2.700, A 0.000, B 0.000, C 0.000} C_DIS
   $VEL.CP = 0.060
   LIN  {X 9.039, Y -1.968, Z 2.700, A 0.000, B 0.000, C 0.000} C_DIS
   $VEL.CP = 0.060
   LIN  {X 9.039, Y 1.968, Z 2.700, A 0.000, B 0.000, C 0.000} C_DIS
   $VEL.CP = 0.060
   LIN  {X -1.968, Y -9.039, Z 2.700, A 0.000, B 0.000, C 0.000} C_DIS
   $VEL.CP = 0.060
   LIN  {X -5.102, Y -9.039, Z 2.700, A 0.000, B 0.000, C 0.000} C_DIS
   $VEL.CP = 0.060
   LIN  {X -9.039, Y -5.102, Z 2.700, A 0.000, B 0.000, C 0.000} C_DIS
   $VEL.CP = 0.060
   LIN  {X -9.039, Y -9.039, Z 2.700, A 0.000, B 0.000, C 0.000} C_DIS
   $VEL.CP = 0.060
   LIN  {X 9.039, Y 9.039, Z 2.700, A 0.000, B 0.000, C 0.000} C_DIS
   $VEL.CP = 0.060
   LIN  {X 9.040, Y 9.040, Z 2.700, A 0.000, B 0.000, C 0.000} C_DIS
   $VEL.CP = 0.060
   LIN  {X 9.039, Y 5.102, Z 2.700, A 0.000, B 0.000, C 0.000} C_DIS
   $VEL.CP = 0.060
   LIN  {X 5.102, Y 9.039, Z 2.700, A 0.000, B 0.000, C 0.000} C_DIS
   $VEL.CP = 0.060
   LIN  {X 1.968, Y 9.039, Z 2.700, A 0.000, B 0.000, C 0.000} C_DIS
   $VEL.CP = 0.060
   LIN  {X -9.039, Y -1.968, Z 2.700, A 0.000, B 0.000, C 0.000} C_DIS
   $VEL.CP = 0.060
   LIN  {X -9.039, Y 1.968, Z 2.700, A 0.000, B 0.000, C 0.000} C_DIS
   $VEL.CP = 0.060
   LIN  {X 1.968, Y -9.039, Z 2.700, A 0.000, B 0.000, C 0.000} C_DIS
   $VEL.CP = 0.060
   LIN  {X 9.040, Y -9.040, Z 2.700, A 0.000, B 0.000, C 0.000} C_DIS

;FOLD ARCOFF WDAT2 LIN P4 CPDAT2 Tool[1]:cmttorch Base[1]:vrashatel ;%{PE}
  ;FOLD Parameters ;%{h}
    ;Params IlfProvider=kukaroboter.arctech.arcofflin; Kuka.IsGlobalPoint=False; Kuka.PointName=P4; Kuka.BlendingEnabled=False; Kuka.MoveDataName=CPDAT2; Kuka.VelocityPath=0.01; Kuka.CurrentCDSetIndex=0; Kuka.MovementParameterFieldEnabled=True; ArcTech.WdatVarName=WDAT2; ArcTech.Basic=3.4.3.1264
  ;ENDFOLD
  $BWDSTART = FALSE
  LDAT_ACT = LCPDAT2
  FDAT_ACT = FP4
  BAS(#CP_PARAMS, gArcBasVelDefinition)
  SET_CD_PARAMS (0)
  TRIGGER WHEN PATH = ArcGetPath(#ArcOffBefore, WDAT2) DELAY = 0 DO ArcMainNG(#ArcOffBeforeOffStd, WDAT2, WP4) PRIO = -1
  TRIGGER WHEN PATH = ArcGetPath(#OnTheFlyArcOff, WDAT2) DELAY = 0 DO ArcMainNG(#ArcOffMoveStd, WDAT2, WP4) PRIO = -1
  ArcMainNG(#ArcOffBeforeMoveStd, WDAT2, WP4)
  LIN XP4
  ArcMainNG(#ArcOffAfterMoveStd, WDAT2, WP4)
;ENDFOLD
   $VEL.CP = 0.080
   LIN  {X 9.039, Y -9.039, Z 2.700, A 0.000, B 0.000, C 0.000} C_DIS

;FOLD ARCON WDAT1 LIN P3 Vel=0.5 m/s CPDAT1 Tool[1]:cmttorch Base[1]:vrashatel ;%{PE}
  ;FOLD Parameters ;%{h}
    ;Params IlfProvider=kukaroboter.arctech.arconlin; Kuka.IsGlobalPoint=False; Kuka.PointName=P3; Kuka.BlendingEnabled=False; Kuka.MoveDataName=CPDAT1; Kuka.VelocityPath=0.5; Kuka.CurrentCDSetIndex=0; Kuka.MovementParameterFieldEnabled=True; ArcTech.WdatVarName=WDAT1; ArcTech.Basic=3.4.3.1264
  ;ENDFOLD
  $BWDSTART = FALSE
  LDAT_ACT = LCPDAT1
  FDAT_ACT = FP3
  BAS(#CP_PARAMS, 0.5)
  SET_CD_PARAMS (0)
  TRIGGER WHEN DISTANCE = 1 DELAY = ArcGetDelay(#PreDefinition, WDAT1) DO ArcMainNG(#PreDefinition, WDAT1, WP3) PRIO = -1
  TRIGGER WHEN PATH = ArcGetPath(#OnTheFlyArcOn, WDAT1) DELAY = ArcGetDelay(#GasPreflow, WDAT1) DO ArcMainNG(#GasPreflow, WDAT1, WP3) PRIO = -1
  TRIGGER WHEN PATH = ArcGetPath(#OnTheFlyArcOn, WDAT1) DELAY = 0 DO ArcMainNG(#ArcOnMoveStd, WDAT1, WP3) PRIO = -1
  ArcMainNG(#ArcOnBeforeMoveStd, WDAT1, WP3)
  LIN XP3
  ArcMainNG(#ArcOnAfterMoveStd, WDAT1, WP3)
;ENDFOLD
   $VEL.CP = 0.060
   LIN  {X -9.039, Y 9.039, Z 2.700, A 0.000, B 0.000, C 0.000} C_DIS
   $VEL.CP = 0.060
   LIN  {X -9.040, Y 9.040, Z 2.700, A 0.000, B 0.000, C 0.000} C_DIS

;FOLD ARCOFF WDAT2 LIN P4 CPDAT2 Tool[1]:cmttorch Base[1]:vrashatel ;%{PE}
  ;FOLD Parameters ;%{h}
    ;Params IlfProvider=kukaroboter.arctech.arcofflin; Kuka.IsGlobalPoint=False; Kuka.PointName=P4; Kuka.BlendingEnabled=False; Kuka.MoveDataName=CPDAT2; Kuka.VelocityPath=0.01; Kuka.CurrentCDSetIndex=0; Kuka.MovementParameterFieldEnabled=True; ArcTech.WdatVarName=WDAT2; ArcTech.Basic=3.4.3.1264
  ;ENDFOLD
  $BWDSTART = FALSE
  LDAT_ACT = LCPDAT2
  FDAT_ACT = FP4
  BAS(#CP_PARAMS, gArcBasVelDefinition)
  SET_CD_PARAMS (0)
  TRIGGER WHEN PATH = ArcGetPath(#ArcOffBefore, WDAT2) DELAY = 0 DO ArcMainNG(#ArcOffBeforeOffStd, WDAT2, WP4) PRIO = -1
  TRIGGER WHEN PATH = ArcGetPath(#OnTheFlyArcOff, WDAT2) DELAY = 0 DO ArcMainNG(#ArcOffMoveStd, WDAT2, WP4) PRIO = -1
  ArcMainNG(#ArcOffBeforeMoveStd, WDAT2, WP4)
  LIN XP4
  ArcMainNG(#ArcOffAfterMoveStd, WDAT2, WP4)
;ENDFOLD
   $VEL.CP = 0.080
   LIN  {X 5.102, Y -9.039, Z 2.700, A 0.000, B 0.000, C 0.000} C_DIS

;FOLD ARCON WDAT1 LIN P3 Vel=0.5 m/s CPDAT1 Tool[1]:cmttorch Base[1]:vrashatel ;%{PE}
  ;FOLD Parameters ;%{h}
    ;Params IlfProvider=kukaroboter.arctech.arconlin; Kuka.IsGlobalPoint=False; Kuka.PointName=P3; Kuka.BlendingEnabled=False; Kuka.MoveDataName=CPDAT1; Kuka.VelocityPath=0.5; Kuka.CurrentCDSetIndex=0; Kuka.MovementParameterFieldEnabled=True; ArcTech.WdatVarName=WDAT1; ArcTech.Basic=3.4.3.1264
  ;ENDFOLD
  $BWDSTART = FALSE
  LDAT_ACT = LCPDAT1
  FDAT_ACT = FP3
  BAS(#CP_PARAMS, 0.5)
  SET_CD_PARAMS (0)
  TRIGGER WHEN DISTANCE = 1 DELAY = ArcGetDelay(#PreDefinition, WDAT1) DO ArcMainNG(#PreDefinition, WDAT1, WP3) PRIO = -1
  TRIGGER WHEN PATH = ArcGetPath(#OnTheFlyArcOn, WDAT1) DELAY = ArcGetDelay(#GasPreflow, WDAT1) DO ArcMainNG(#GasPreflow, WDAT1, WP3) PRIO = -1
  TRIGGER WHEN PATH = ArcGetPath(#OnTheFlyArcOn, WDAT1) DELAY = 0 DO ArcMainNG(#ArcOnMoveStd, WDAT1, WP3) PRIO = -1
  ArcMainNG(#ArcOnBeforeMoveStd, WDAT1, WP3)
  LIN XP3
  ArcMainNG(#ArcOnAfterMoveStd, WDAT1, WP3)
;ENDFOLD
   $VEL.CP = 0.025
   LIN  {X 5.102, Y -9.039, Z 2.700, A 0.000, B 0.000, C 0.000} C_DIS
   $VEL.CP = 0.060
   LIN  {X 9.039, Y -5.102, Z 2.700, A 0.000, B 0.000, C 0.000} C_DIS
   $VEL.CP = 0.060
   LIN  {X 9.039, Y -9.039, Z 2.700, A 0.000, B 0.000, C 0.000} C_DIS

;FOLD ARCOFF WDAT2 LIN P4 CPDAT2 Tool[1]:cmttorch Base[1]:vrashatel ;%{PE}
  ;FOLD Parameters ;%{h}
    ;Params IlfProvider=kukaroboter.arctech.arcofflin; Kuka.IsGlobalPoint=False; Kuka.PointName=P4; Kuka.BlendingEnabled=False; Kuka.MoveDataName=CPDAT2; Kuka.VelocityPath=0.01; Kuka.CurrentCDSetIndex=0; Kuka.MovementParameterFieldEnabled=True; ArcTech.WdatVarName=WDAT2; ArcTech.Basic=3.4.3.1264
  ;ENDFOLD
  $BWDSTART = FALSE
  LDAT_ACT = LCPDAT2
  FDAT_ACT = FP4
  BAS(#CP_PARAMS, gArcBasVelDefinition)
  SET_CD_PARAMS (0)
  TRIGGER WHEN PATH = ArcGetPath(#ArcOffBefore, WDAT2) DELAY = 0 DO ArcMainNG(#ArcOffBeforeOffStd, WDAT2, WP4) PRIO = -1
  TRIGGER WHEN PATH = ArcGetPath(#OnTheFlyArcOff, WDAT2) DELAY = 0 DO ArcMainNG(#ArcOffMoveStd, WDAT2, WP4) PRIO = -1
  ArcMainNG(#ArcOffBeforeMoveStd, WDAT2, WP4)
  LIN XP4
  ArcMainNG(#ArcOffAfterMoveStd, WDAT2, WP4)
;ENDFOLD
   $VEL.CP = 0.060
   LIN  {X 9.039, Y -9.139, Z 2.700, A 0.000, B 0.000, C 0.000} C_DIS
   $VEL.CP = 0.010
   LIN  {X 9.039, Y -9.139, Z 2.900, A 0.000, B 0.000, C 0.000} C_DIS
   $VEL.CP = 0.080
   LIN  {X -9.530, Y 9.530, Z 2.900, A 0.000, B 0.000, C 0.000} C_DIS
   $VEL.CP = 0.080
   LIN  {X -9.800, Y 9.800, Z 2.900, A 0.000, B 0.000, C 0.000} C_DIS

;FOLD ARCON WDAT1 LIN P3 Vel=0.5 m/s CPDAT1 Tool[1]:cmttorch Base[1]:vrashatel ;%{PE}
  ;FOLD Parameters ;%{h}
    ;Params IlfProvider=kukaroboter.arctech.arconlin; Kuka.IsGlobalPoint=False; Kuka.PointName=P3; Kuka.BlendingEnabled=False; Kuka.MoveDataName=CPDAT1; Kuka.VelocityPath=0.5; Kuka.CurrentCDSetIndex=0; Kuka.MovementParameterFieldEnabled=True; ArcTech.WdatVarName=WDAT1; ArcTech.Basic=3.4.3.1264
  ;ENDFOLD
  $BWDSTART = FALSE
  LDAT_ACT = LCPDAT1
  FDAT_ACT = FP3
  BAS(#CP_PARAMS, 0.5)
  SET_CD_PARAMS (0)
  TRIGGER WHEN DISTANCE = 1 DELAY = ArcGetDelay(#PreDefinition, WDAT1) DO ArcMainNG(#PreDefinition, WDAT1, WP3) PRIO = -1
  TRIGGER WHEN PATH = ArcGetPath(#OnTheFlyArcOn, WDAT1) DELAY = ArcGetDelay(#GasPreflow, WDAT1) DO ArcMainNG(#GasPreflow, WDAT1, WP3) PRIO = -1
  TRIGGER WHEN PATH = ArcGetPath(#OnTheFlyArcOn, WDAT1) DELAY = 0 DO ArcMainNG(#ArcOnMoveStd, WDAT1, WP3) PRIO = -1
  ArcMainNG(#ArcOnBeforeMoveStd, WDAT1, WP3)
  LIN XP3
  ArcMainNG(#ArcOnAfterMoveStd, WDAT1, WP3)
;ENDFOLD
   $VEL.CP = 0.025
   LIN  {X -9.800, Y 9.800, Z 2.900, A 0.000, B 0.000, C 0.000} C_DIS
   $VEL.CP = 0.060
   LIN  {X -9.800, Y -9.800, Z 2.900, A 0.000, B 0.000, C 0.000} C_DIS
   $VEL.CP = 0.060
   LIN  {X 9.800, Y -9.800, Z 2.900, A 0.000, B 0.000, C 0.000} C_DIS
   $VEL.CP = 0.060
   LIN  {X 9.800, Y 9.800, Z 2.900, A 0.000, B 0.000, C 0.000} C_DIS
   $VEL.CP = 0.060
   LIN  {X -9.800, Y 9.800, Z 2.900, A 0.000, B 0.000, C 0.000} C_DIS

;FOLD ARCOFF WDAT2 LIN P4 CPDAT2 Tool[1]:cmttorch Base[1]:vrashatel ;%{PE}
  ;FOLD Parameters ;%{h}
    ;Params IlfProvider=kukaroboter.arctech.arcofflin; Kuka.IsGlobalPoint=False; Kuka.PointName=P4; Kuka.BlendingEnabled=False; Kuka.MoveDataName=CPDAT2; Kuka.VelocityPath=0.01; Kuka.CurrentCDSetIndex=0; Kuka.MovementParameterFieldEnabled=True; ArcTech.WdatVarName=WDAT2; ArcTech.Basic=3.4.3.1264
  ;ENDFOLD
  $BWDSTART = FALSE
  LDAT_ACT = LCPDAT2
  FDAT_ACT = FP4
  BAS(#CP_PARAMS, gArcBasVelDefinition)
  SET_CD_PARAMS (0)
  TRIGGER WHEN PATH = ArcGetPath(#ArcOffBefore, WDAT2) DELAY = 0 DO ArcMainNG(#ArcOffBeforeOffStd, WDAT2, WP4) PRIO = -1
  TRIGGER WHEN PATH = ArcGetPath(#OnTheFlyArcOff, WDAT2) DELAY = 0 DO ArcMainNG(#ArcOffMoveStd, WDAT2, WP4) PRIO = -1
  ArcMainNG(#ArcOffBeforeMoveStd, WDAT2, WP4)
  LIN XP4
  ArcMainNG(#ArcOffAfterMoveStd, WDAT2, WP4)
;ENDFOLD
   $VEL.CP = 0.080
   LIN  {X -9.800, Y 9.600, Z 2.900, A 0.000, B 0.000, C 0.000} C_DIS
   $VEL.CP = 0.080
   LIN  {X -9.360, Y 9.360, Z 2.900, A 0.000, B 0.000, C 0.000} C_DIS
   $VEL.CP = 0.080
   LIN  {X -9.400, Y 9.400, Z 2.900, A 0.000, B 0.000, C 0.000} C_DIS

;FOLD ARCON WDAT1 LIN P3 Vel=0.5 m/s CPDAT1 Tool[1]:cmttorch Base[1]:vrashatel ;%{PE}
  ;FOLD Parameters ;%{h}
    ;Params IlfProvider=kukaroboter.arctech.arconlin; Kuka.IsGlobalPoint=False; Kuka.PointName=P3; Kuka.BlendingEnabled=False; Kuka.MoveDataName=CPDAT1; Kuka.VelocityPath=0.5; Kuka.CurrentCDSetIndex=0; Kuka.MovementParameterFieldEnabled=True; ArcTech.WdatVarName=WDAT1; ArcTech.Basic=3.4.3.1264
  ;ENDFOLD
  $BWDSTART = FALSE
  LDAT_ACT = LCPDAT1
  FDAT_ACT = FP3
  BAS(#CP_PARAMS, 0.5)
  SET_CD_PARAMS (0)
  TRIGGER WHEN DISTANCE = 1 DELAY = ArcGetDelay(#PreDefinition, WDAT1) DO ArcMainNG(#PreDefinition, WDAT1, WP3) PRIO = -1
  TRIGGER WHEN PATH = ArcGetPath(#OnTheFlyArcOn, WDAT1) DELAY = ArcGetDelay(#GasPreflow, WDAT1) DO ArcMainNG(#GasPreflow, WDAT1, WP3) PRIO = -1
  TRIGGER WHEN PATH = ArcGetPath(#OnTheFlyArcOn, WDAT1) DELAY = 0 DO ArcMainNG(#ArcOnMoveStd, WDAT1, WP3) PRIO = -1
  ArcMainNG(#ArcOnBeforeMoveStd, WDAT1, WP3)
  LIN XP3
  ArcMainNG(#ArcOnAfterMoveStd, WDAT1, WP3)
;ENDFOLD
   $VEL.CP = 0.060
   LIN  {X -9.400, Y -9.400, Z 2.900, A 0.000, B 0.000, C 0.000} C_DIS
   $VEL.CP = 0.060
   LIN  {X 9.400, Y -9.400, Z 2.900, A 0.000, B 0.000, C 0.000} C_DIS
   $VEL.CP = 0.060
   LIN  {X 9.400, Y 9.400, Z 2.900, A 0.000, B 0.000, C 0.000} C_DIS
   $VEL.CP = 0.060
   LIN  {X -9.400, Y 9.400, Z 2.900, A 0.000, B 0.000, C 0.000} C_DIS

;FOLD ARCOFF WDAT2 LIN P4 CPDAT2 Tool[1]:cmttorch Base[1]:vrashatel ;%{PE}
  ;FOLD Parameters ;%{h}
    ;Params IlfProvider=kukaroboter.arctech.arcofflin; Kuka.IsGlobalPoint=False; Kuka.PointName=P4; Kuka.BlendingEnabled=False; Kuka.MoveDataName=CPDAT2; Kuka.VelocityPath=0.01; Kuka.CurrentCDSetIndex=0; Kuka.MovementParameterFieldEnabled=True; ArcTech.WdatVarName=WDAT2; ArcTech.Basic=3.4.3.1264
  ;ENDFOLD
  $BWDSTART = FALSE
  LDAT_ACT = LCPDAT2
  FDAT_ACT = FP4
  BAS(#CP_PARAMS, gArcBasVelDefinition)
  SET_CD_PARAMS (0)
  TRIGGER WHEN PATH = ArcGetPath(#ArcOffBefore, WDAT2) DELAY = 0 DO ArcMainNG(#ArcOffBeforeOffStd, WDAT2, WP4) PRIO = -1
  TRIGGER WHEN PATH = ArcGetPath(#OnTheFlyArcOff, WDAT2) DELAY = 0 DO ArcMainNG(#ArcOffMoveStd, WDAT2, WP4) PRIO = -1
  ArcMainNG(#ArcOffBeforeMoveStd, WDAT2, WP4)
  LIN XP4
  ArcMainNG(#ArcOffAfterMoveStd, WDAT2, WP4)
;ENDFOLD
   $VEL.CP = 0.080
   LIN  {X -9.040, Y 9.040, Z 2.900, A 0.000, B 0.000, C 0.000} C_DIS

;FOLD ARCON WDAT1 LIN P3 Vel=0.5 m/s CPDAT1 Tool[1]:cmttorch Base[1]:vrashatel ;%{PE}
  ;FOLD Parameters ;%{h}
    ;Params IlfProvider=kukaroboter.arctech.arconlin; Kuka.IsGlobalPoint=False; Kuka.PointName=P3; Kuka.BlendingEnabled=False; Kuka.MoveDataName=CPDAT1; Kuka.VelocityPath=0.5; Kuka.CurrentCDSetIndex=0; Kuka.MovementParameterFieldEnabled=True; ArcTech.WdatVarName=WDAT1; ArcTech.Basic=3.4.3.1264
  ;ENDFOLD
  $BWDSTART = FALSE
  LDAT_ACT = LCPDAT1
  FDAT_ACT = FP3
  BAS(#CP_PARAMS, 0.5)
  SET_CD_PARAMS (0)
  TRIGGER WHEN DISTANCE = 1 DELAY = ArcGetDelay(#PreDefinition, WDAT1) DO ArcMainNG(#PreDefinition, WDAT1, WP3) PRIO = -1
  TRIGGER WHEN PATH = ArcGetPath(#OnTheFlyArcOn, WDAT1) DELAY = ArcGetDelay(#GasPreflow, WDAT1) DO ArcMainNG(#GasPreflow, WDAT1, WP3) PRIO = -1
  TRIGGER WHEN PATH = ArcGetPath(#OnTheFlyArcOn, WDAT1) DELAY = 0 DO ArcMainNG(#ArcOnMoveStd, WDAT1, WP3) PRIO = -1
  ArcMainNG(#ArcOnBeforeMoveStd, WDAT1, WP3)
  LIN XP3
  ArcMainNG(#ArcOnAfterMoveStd, WDAT1, WP3)
;ENDFOLD
   $VEL.CP = 0.060
   LIN  {X -9.039, Y 5.102, Z 2.900, A 0.000, B 0.000, C 0.000} C_DIS
   $VEL.CP = 0.060
   LIN  {X -5.102, Y 9.039, Z 2.900, A 0.000, B 0.000, C 0.000} C_DIS
   $VEL.CP = 0.060
   LIN  {X -1.968, Y 9.039, Z 2.900, A 0.000, B 0.000, C 0.000} C_DIS
   $VEL.CP = 0.060
   LIN  {X 9.039, Y -1.968, Z 2.900, A 0.000, B 0.000, C 0.000} C_DIS
   $VEL.CP = 0.060
   LIN  {X 9.039, Y 1.968, Z 2.900, A 0.000, B 0.000, C 0.000} C_DIS
   $VEL.CP = 0.060
   LIN  {X -1.968, Y -9.039, Z 2.900, A 0.000, B 0.000, C 0.000} C_DIS
   $VEL.CP = 0.060
   LIN  {X -5.102, Y -9.039, Z 2.900, A 0.000, B 0.000, C 0.000} C_DIS
   $VEL.CP = 0.060
   LIN  {X -9.039, Y -5.102, Z 2.900, A 0.000, B 0.000, C 0.000} C_DIS
   $VEL.CP = 0.060
   LIN  {X -9.039, Y -9.039, Z 2.900, A 0.000, B 0.000, C 0.000} C_DIS
   $VEL.CP = 0.060
   LIN  {X 9.039, Y 9.039, Z 2.900, A 0.000, B 0.000, C 0.000} C_DIS
   $VEL.CP = 0.060
   LIN  {X 9.040, Y 9.040, Z 2.900, A 0.000, B 0.000, C 0.000} C_DIS
   $VEL.CP = 0.060
   LIN  {X 9.039, Y 5.102, Z 2.900, A 0.000, B 0.000, C 0.000} C_DIS
   $VEL.CP = 0.060
   LIN  {X 5.102, Y 9.039, Z 2.900, A 0.000, B 0.000, C 0.000} C_DIS
   $VEL.CP = 0.060
   LIN  {X 1.968, Y 9.039, Z 2.900, A 0.000, B 0.000, C 0.000} C_DIS
   $VEL.CP = 0.060
   LIN  {X -9.039, Y -1.968, Z 2.900, A 0.000, B 0.000, C 0.000} C_DIS
   $VEL.CP = 0.060
   LIN  {X -9.039, Y 1.968, Z 2.900, A 0.000, B 0.000, C 0.000} C_DIS
   $VEL.CP = 0.060
   LIN  {X 1.968, Y -9.039, Z 2.900, A 0.000, B 0.000, C 0.000} C_DIS
   $VEL.CP = 0.060
   LIN  {X 9.040, Y -9.040, Z 2.900, A 0.000, B 0.000, C 0.000} C_DIS

;FOLD ARCOFF WDAT2 LIN P4 CPDAT2 Tool[1]:cmttorch Base[1]:vrashatel ;%{PE}
  ;FOLD Parameters ;%{h}
    ;Params IlfProvider=kukaroboter.arctech.arcofflin; Kuka.IsGlobalPoint=False; Kuka.PointName=P4; Kuka.BlendingEnabled=False; Kuka.MoveDataName=CPDAT2; Kuka.VelocityPath=0.01; Kuka.CurrentCDSetIndex=0; Kuka.MovementParameterFieldEnabled=True; ArcTech.WdatVarName=WDAT2; ArcTech.Basic=3.4.3.1264
  ;ENDFOLD
  $BWDSTART = FALSE
  LDAT_ACT = LCPDAT2
  FDAT_ACT = FP4
  BAS(#CP_PARAMS, gArcBasVelDefinition)
  SET_CD_PARAMS (0)
  TRIGGER WHEN PATH = ArcGetPath(#ArcOffBefore, WDAT2) DELAY = 0 DO ArcMainNG(#ArcOffBeforeOffStd, WDAT2, WP4) PRIO = -1
  TRIGGER WHEN PATH = ArcGetPath(#OnTheFlyArcOff, WDAT2) DELAY = 0 DO ArcMainNG(#ArcOffMoveStd, WDAT2, WP4) PRIO = -1
  ArcMainNG(#ArcOffBeforeMoveStd, WDAT2, WP4)
  LIN XP4
  ArcMainNG(#ArcOffAfterMoveStd, WDAT2, WP4)
;ENDFOLD
   $VEL.CP = 0.080
   LIN  {X 9.039, Y -9.039, Z 2.900, A 0.000, B 0.000, C 0.000} C_DIS

;FOLD ARCON WDAT1 LIN P3 Vel=0.5 m/s CPDAT1 Tool[1]:cmttorch Base[1]:vrashatel ;%{PE}
  ;FOLD Parameters ;%{h}
    ;Params IlfProvider=kukaroboter.arctech.arconlin; Kuka.IsGlobalPoint=False; Kuka.PointName=P3; Kuka.BlendingEnabled=False; Kuka.MoveDataName=CPDAT1; Kuka.VelocityPath=0.5; Kuka.CurrentCDSetIndex=0; Kuka.MovementParameterFieldEnabled=True; ArcTech.WdatVarName=WDAT1; ArcTech.Basic=3.4.3.1264
  ;ENDFOLD
  $BWDSTART = FALSE
  LDAT_ACT = LCPDAT1
  FDAT_ACT = FP3
  BAS(#CP_PARAMS, 0.5)
  SET_CD_PARAMS (0)
  TRIGGER WHEN DISTANCE = 1 DELAY = ArcGetDelay(#PreDefinition, WDAT1) DO ArcMainNG(#PreDefinition, WDAT1, WP3) PRIO = -1
  TRIGGER WHEN PATH = ArcGetPath(#OnTheFlyArcOn, WDAT1) DELAY = ArcGetDelay(#GasPreflow, WDAT1) DO ArcMainNG(#GasPreflow, WDAT1, WP3) PRIO = -1
  TRIGGER WHEN PATH = ArcGetPath(#OnTheFlyArcOn, WDAT1) DELAY = 0 DO ArcMainNG(#ArcOnMoveStd, WDAT1, WP3) PRIO = -1
  ArcMainNG(#ArcOnBeforeMoveStd, WDAT1, WP3)
  LIN XP3
  ArcMainNG(#ArcOnAfterMoveStd, WDAT1, WP3)
;ENDFOLD
   $VEL.CP = 0.060
   LIN  {X -9.039, Y 9.039, Z 2.900, A 0.000, B 0.000, C 0.000} C_DIS
   $VEL.CP = 0.060
   LIN  {X -9.040, Y 9.040, Z 2.900, A 0.000, B 0.000, C 0.000} C_DIS

;FOLD ARCOFF WDAT2 LIN P4 CPDAT2 Tool[1]:cmttorch Base[1]:vrashatel ;%{PE}
  ;FOLD Parameters ;%{h}
    ;Params IlfProvider=kukaroboter.arctech.arcofflin; Kuka.IsGlobalPoint=False; Kuka.PointName=P4; Kuka.BlendingEnabled=False; Kuka.MoveDataName=CPDAT2; Kuka.VelocityPath=0.01; Kuka.CurrentCDSetIndex=0; Kuka.MovementParameterFieldEnabled=True; ArcTech.WdatVarName=WDAT2; ArcTech.Basic=3.4.3.1264
  ;ENDFOLD
  $BWDSTART = FALSE
  LDAT_ACT = LCPDAT2
  FDAT_ACT = FP4
  BAS(#CP_PARAMS, gArcBasVelDefinition)
  SET_CD_PARAMS (0)
  TRIGGER WHEN PATH = ArcGetPath(#ArcOffBefore, WDAT2) DELAY = 0 DO ArcMainNG(#ArcOffBeforeOffStd, WDAT2, WP4) PRIO = -1
  TRIGGER WHEN PATH = ArcGetPath(#OnTheFlyArcOff, WDAT2) DELAY = 0 DO ArcMainNG(#ArcOffMoveStd, WDAT2, WP4) PRIO = -1
  ArcMainNG(#ArcOffBeforeMoveStd, WDAT2, WP4)
  LIN XP4
  ArcMainNG(#ArcOffAfterMoveStd, WDAT2, WP4)
;ENDFOLD
   $VEL.CP = 0.080
   LIN  {X 5.102, Y -9.039, Z 2.900, A 0.000, B 0.000, C 0.000} C_DIS

;FOLD ARCON WDAT1 LIN P3 Vel=0.5 m/s CPDAT1 Tool[1]:cmttorch Base[1]:vrashatel ;%{PE}
  ;FOLD Parameters ;%{h}
    ;Params IlfProvider=kukaroboter.arctech.arconlin; Kuka.IsGlobalPoint=False; Kuka.PointName=P3; Kuka.BlendingEnabled=False; Kuka.MoveDataName=CPDAT1; Kuka.VelocityPath=0.5; Kuka.CurrentCDSetIndex=0; Kuka.MovementParameterFieldEnabled=True; ArcTech.WdatVarName=WDAT1; ArcTech.Basic=3.4.3.1264
  ;ENDFOLD
  $BWDSTART = FALSE
  LDAT_ACT = LCPDAT1
  FDAT_ACT = FP3
  BAS(#CP_PARAMS, 0.5)
  SET_CD_PARAMS (0)
  TRIGGER WHEN DISTANCE = 1 DELAY = ArcGetDelay(#PreDefinition, WDAT1) DO ArcMainNG(#PreDefinition, WDAT1, WP3) PRIO = -1
  TRIGGER WHEN PATH = ArcGetPath(#OnTheFlyArcOn, WDAT1) DELAY = ArcGetDelay(#GasPreflow, WDAT1) DO ArcMainNG(#GasPreflow, WDAT1, WP3) PRIO = -1
  TRIGGER WHEN PATH = ArcGetPath(#OnTheFlyArcOn, WDAT1) DELAY = 0 DO ArcMainNG(#ArcOnMoveStd, WDAT1, WP3) PRIO = -1
  ArcMainNG(#ArcOnBeforeMoveStd, WDAT1, WP3)
  LIN XP3
  ArcMainNG(#ArcOnAfterMoveStd, WDAT1, WP3)
;ENDFOLD
   $VEL.CP = 0.025
   LIN  {X 5.102, Y -9.039, Z 2.900, A 0.000, B 0.000, C 0.000} C_DIS
   $VEL.CP = 0.060
   LIN  {X 9.039, Y -5.102, Z 2.900, A 0.000, B 0.000, C 0.000} C_DIS
   $VEL.CP = 0.060
   LIN  {X 9.039, Y -9.039, Z 2.900, A 0.000, B 0.000, C 0.000} C_DIS

;FOLD ARCOFF WDAT2 LIN P4 CPDAT2 Tool[1]:cmttorch Base[1]:vrashatel ;%{PE}
  ;FOLD Parameters ;%{h}
    ;Params IlfProvider=kukaroboter.arctech.arcofflin; Kuka.IsGlobalPoint=False; Kuka.PointName=P4; Kuka.BlendingEnabled=False; Kuka.MoveDataName=CPDAT2; Kuka.VelocityPath=0.01; Kuka.CurrentCDSetIndex=0; Kuka.MovementParameterFieldEnabled=True; ArcTech.WdatVarName=WDAT2; ArcTech.Basic=3.4.3.1264
  ;ENDFOLD
  $BWDSTART = FALSE
  LDAT_ACT = LCPDAT2
  FDAT_ACT = FP4
  BAS(#CP_PARAMS, gArcBasVelDefinition)
  SET_CD_PARAMS (0)
  TRIGGER WHEN PATH = ArcGetPath(#ArcOffBefore, WDAT2) DELAY = 0 DO ArcMainNG(#ArcOffBeforeOffStd, WDAT2, WP4) PRIO = -1
  TRIGGER WHEN PATH = ArcGetPath(#OnTheFlyArcOff, WDAT2) DELAY = 0 DO ArcMainNG(#ArcOffMoveStd, WDAT2, WP4) PRIO = -1
  ArcMainNG(#ArcOffBeforeMoveStd, WDAT2, WP4)
  LIN XP4
  ArcMainNG(#ArcOffAfterMoveStd, WDAT2, WP4)
;ENDFOLD
   $VEL.CP = 0.060
   LIN  {X 9.039, Y -9.139, Z 2.900, A 0.000, B 0.000, C 0.000} C_DIS
   $VEL.CP = 0.010
   LIN  {X 9.039, Y -9.139, Z 3.100, A 0.000, B 0.000, C 0.000} C_DIS
   $VEL.CP = 0.080
   LIN  {X -9.530, Y 9.530, Z 3.100, A 0.000, B 0.000, C 0.000} C_DIS
   $VEL.CP = 0.080
   LIN  {X -9.800, Y 9.800, Z 3.100, A 0.000, B 0.000, C 0.000} C_DIS

;FOLD ARCON WDAT1 LIN P3 Vel=0.5 m/s CPDAT1 Tool[1]:cmttorch Base[1]:vrashatel ;%{PE}
  ;FOLD Parameters ;%{h}
    ;Params IlfProvider=kukaroboter.arctech.arconlin; Kuka.IsGlobalPoint=False; Kuka.PointName=P3; Kuka.BlendingEnabled=False; Kuka.MoveDataName=CPDAT1; Kuka.VelocityPath=0.5; Kuka.CurrentCDSetIndex=0; Kuka.MovementParameterFieldEnabled=True; ArcTech.WdatVarName=WDAT1; ArcTech.Basic=3.4.3.1264
  ;ENDFOLD
  $BWDSTART = FALSE
  LDAT_ACT = LCPDAT1
  FDAT_ACT = FP3
  BAS(#CP_PARAMS, 0.5)
  SET_CD_PARAMS (0)
  TRIGGER WHEN DISTANCE = 1 DELAY = ArcGetDelay(#PreDefinition, WDAT1) DO ArcMainNG(#PreDefinition, WDAT1, WP3) PRIO = -1
  TRIGGER WHEN PATH = ArcGetPath(#OnTheFlyArcOn, WDAT1) DELAY = ArcGetDelay(#GasPreflow, WDAT1) DO ArcMainNG(#GasPreflow, WDAT1, WP3) PRIO = -1
  TRIGGER WHEN PATH = ArcGetPath(#OnTheFlyArcOn, WDAT1) DELAY = 0 DO ArcMainNG(#ArcOnMoveStd, WDAT1, WP3) PRIO = -1
  ArcMainNG(#ArcOnBeforeMoveStd, WDAT1, WP3)
  LIN XP3
  ArcMainNG(#ArcOnAfterMoveStd, WDAT1, WP3)
;ENDFOLD
   $VEL.CP = 0.025
   LIN  {X -9.800, Y 9.800, Z 3.100, A 0.000, B 0.000, C 0.000} C_DIS
   $VEL.CP = 0.060
   LIN  {X -9.800, Y -9.800, Z 3.100, A 0.000, B 0.000, C 0.000} C_DIS
   $VEL.CP = 0.060
   LIN  {X 9.800, Y -9.800, Z 3.100, A 0.000, B 0.000, C 0.000} C_DIS
   $VEL.CP = 0.060
   LIN  {X 9.800, Y 9.800, Z 3.100, A 0.000, B 0.000, C 0.000} C_DIS
   $VEL.CP = 0.060
   LIN  {X -9.800, Y 9.800, Z 3.100, A 0.000, B 0.000, C 0.000} C_DIS

;FOLD ARCOFF WDAT2 LIN P4 CPDAT2 Tool[1]:cmttorch Base[1]:vrashatel ;%{PE}
  ;FOLD Parameters ;%{h}
    ;Params IlfProvider=kukaroboter.arctech.arcofflin; Kuka.IsGlobalPoint=False; Kuka.PointName=P4; Kuka.BlendingEnabled=False; Kuka.MoveDataName=CPDAT2; Kuka.VelocityPath=0.01; Kuka.CurrentCDSetIndex=0; Kuka.MovementParameterFieldEnabled=True; ArcTech.WdatVarName=WDAT2; ArcTech.Basic=3.4.3.1264
  ;ENDFOLD
  $BWDSTART = FALSE
  LDAT_ACT = LCPDAT2
  FDAT_ACT = FP4
  BAS(#CP_PARAMS, gArcBasVelDefinition)
  SET_CD_PARAMS (0)
  TRIGGER WHEN PATH = ArcGetPath(#ArcOffBefore, WDAT2) DELAY = 0 DO ArcMainNG(#ArcOffBeforeOffStd, WDAT2, WP4) PRIO = -1
  TRIGGER WHEN PATH = ArcGetPath(#OnTheFlyArcOff, WDAT2) DELAY = 0 DO ArcMainNG(#ArcOffMoveStd, WDAT2, WP4) PRIO = -1
  ArcMainNG(#ArcOffBeforeMoveStd, WDAT2, WP4)
  LIN XP4
  ArcMainNG(#ArcOffAfterMoveStd, WDAT2, WP4)
;ENDFOLD
   $VEL.CP = 0.080
   LIN  {X -9.800, Y 9.600, Z 3.100, A 0.000, B 0.000, C 0.000} C_DIS
   $VEL.CP = 0.080
   LIN  {X -9.360, Y 9.360, Z 3.100, A 0.000, B 0.000, C 0.000} C_DIS
   $VEL.CP = 0.080
   LIN  {X -9.400, Y 9.400, Z 3.100, A 0.000, B 0.000, C 0.000} C_DIS

;FOLD ARCON WDAT1 LIN P3 Vel=0.5 m/s CPDAT1 Tool[1]:cmttorch Base[1]:vrashatel ;%{PE}
  ;FOLD Parameters ;%{h}
    ;Params IlfProvider=kukaroboter.arctech.arconlin; Kuka.IsGlobalPoint=False; Kuka.PointName=P3; Kuka.BlendingEnabled=False; Kuka.MoveDataName=CPDAT1; Kuka.VelocityPath=0.5; Kuka.CurrentCDSetIndex=0; Kuka.MovementParameterFieldEnabled=True; ArcTech.WdatVarName=WDAT1; ArcTech.Basic=3.4.3.1264
  ;ENDFOLD
  $BWDSTART = FALSE
  LDAT_ACT = LCPDAT1
  FDAT_ACT = FP3
  BAS(#CP_PARAMS, 0.5)
  SET_CD_PARAMS (0)
  TRIGGER WHEN DISTANCE = 1 DELAY = ArcGetDelay(#PreDefinition, WDAT1) DO ArcMainNG(#PreDefinition, WDAT1, WP3) PRIO = -1
  TRIGGER WHEN PATH = ArcGetPath(#OnTheFlyArcOn, WDAT1) DELAY = ArcGetDelay(#GasPreflow, WDAT1) DO ArcMainNG(#GasPreflow, WDAT1, WP3) PRIO = -1
  TRIGGER WHEN PATH = ArcGetPath(#OnTheFlyArcOn, WDAT1) DELAY = 0 DO ArcMainNG(#ArcOnMoveStd, WDAT1, WP3) PRIO = -1
  ArcMainNG(#ArcOnBeforeMoveStd, WDAT1, WP3)
  LIN XP3
  ArcMainNG(#ArcOnAfterMoveStd, WDAT1, WP3)
;ENDFOLD
   $VEL.CP = 0.060
   LIN  {X -9.400, Y -9.400, Z 3.100, A 0.000, B 0.000, C 0.000} C_DIS
   $VEL.CP = 0.060
   LIN  {X 9.400, Y -9.400, Z 3.100, A 0.000, B 0.000, C 0.000} C_DIS
   $VEL.CP = 0.060
   LIN  {X 9.400, Y 9.400, Z 3.100, A 0.000, B 0.000, C 0.000} C_DIS
   $VEL.CP = 0.060
   LIN  {X -9.400, Y 9.400, Z 3.100, A 0.000, B 0.000, C 0.000} C_DIS

;FOLD ARCOFF WDAT2 LIN P4 CPDAT2 Tool[1]:cmttorch Base[1]:vrashatel ;%{PE}
  ;FOLD Parameters ;%{h}
    ;Params IlfProvider=kukaroboter.arctech.arcofflin; Kuka.IsGlobalPoint=False; Kuka.PointName=P4; Kuka.BlendingEnabled=False; Kuka.MoveDataName=CPDAT2; Kuka.VelocityPath=0.01; Kuka.CurrentCDSetIndex=0; Kuka.MovementParameterFieldEnabled=True; ArcTech.WdatVarName=WDAT2; ArcTech.Basic=3.4.3.1264
  ;ENDFOLD
  $BWDSTART = FALSE
  LDAT_ACT = LCPDAT2
  FDAT_ACT = FP4
  BAS(#CP_PARAMS, gArcBasVelDefinition)
  SET_CD_PARAMS (0)
  TRIGGER WHEN PATH = ArcGetPath(#ArcOffBefore, WDAT2) DELAY = 0 DO ArcMainNG(#ArcOffBeforeOffStd, WDAT2, WP4) PRIO = -1
  TRIGGER WHEN PATH = ArcGetPath(#OnTheFlyArcOff, WDAT2) DELAY = 0 DO ArcMainNG(#ArcOffMoveStd, WDAT2, WP4) PRIO = -1
  ArcMainNG(#ArcOffBeforeMoveStd, WDAT2, WP4)
  LIN XP4
  ArcMainNG(#ArcOffAfterMoveStd, WDAT2, WP4)
;ENDFOLD
   $VEL.CP = 0.080
   LIN  {X -9.039, Y 1.968, Z 3.100, A 0.000, B 0.000, C 0.000} C_DIS

;FOLD ARCON WDAT1 LIN P3 Vel=0.5 m/s CPDAT1 Tool[1]:cmttorch Base[1]:vrashatel ;%{PE}
  ;FOLD Parameters ;%{h}
    ;Params IlfProvider=kukaroboter.arctech.arconlin; Kuka.IsGlobalPoint=False; Kuka.PointName=P3; Kuka.BlendingEnabled=False; Kuka.MoveDataName=CPDAT1; Kuka.VelocityPath=0.5; Kuka.CurrentCDSetIndex=0; Kuka.MovementParameterFieldEnabled=True; ArcTech.WdatVarName=WDAT1; ArcTech.Basic=3.4.3.1264
  ;ENDFOLD
  $BWDSTART = FALSE
  LDAT_ACT = LCPDAT1
  FDAT_ACT = FP3
  BAS(#CP_PARAMS, 0.5)
  SET_CD_PARAMS (0)
  TRIGGER WHEN DISTANCE = 1 DELAY = ArcGetDelay(#PreDefinition, WDAT1) DO ArcMainNG(#PreDefinition, WDAT1, WP3) PRIO = -1
  TRIGGER WHEN PATH = ArcGetPath(#OnTheFlyArcOn, WDAT1) DELAY = ArcGetDelay(#GasPreflow, WDAT1) DO ArcMainNG(#GasPreflow, WDAT1, WP3) PRIO = -1
  TRIGGER WHEN PATH = ArcGetPath(#OnTheFlyArcOn, WDAT1) DELAY = 0 DO ArcMainNG(#ArcOnMoveStd, WDAT1, WP3) PRIO = -1
  ArcMainNG(#ArcOnBeforeMoveStd, WDAT1, WP3)
  LIN XP3
  ArcMainNG(#ArcOnAfterMoveStd, WDAT1, WP3)
;ENDFOLD
   $VEL.CP = 0.060
   LIN  {X 1.700, Y -8.771, Z 3.100, A 0.000, B 0.000, C 0.000} C_DIS
   $VEL.CP = 0.060
   LIN  {X 1.699, Y -7.348, Z 3.100, A 0.000, B 0.000, C 0.000} C_DIS
   $VEL.CP = 0.060
   LIN  {X 4.998, Y -7.348, Z 3.100, A 0.000, B 0.000, C 0.000} C_DIS
   $VEL.CP = 0.060
   LIN  {X 5.000, Y -9.040, Z 3.100, A 0.000, B 0.000, C 0.000} C_DIS
   $VEL.CP = 0.060
   LIN  {X 5.103, Y -9.038, Z 3.100, A 0.000, B 0.000, C 0.000} C_DIS
   $VEL.CP = 0.060
   LIN  {X 9.039, Y -5.102, Z 3.100, A 0.000, B 0.000, C 0.000} C_DIS
   $VEL.CP = 0.060
   LIN  {X 9.039, Y -9.039, Z 3.100, A 0.000, B 0.000, C 0.000} C_DIS
   $VEL.CP = 0.060
   LIN  {X -9.039, Y 9.039, Z 3.100, A 0.000, B 0.000, C 0.000} C_DIS
   $VEL.CP = 0.060
   LIN  {X -5.102, Y 9.039, Z 3.100, A 0.000, B 0.000, C 0.000} C_DIS
   $VEL.CP = 0.060
   LIN  {X -9.039, Y 5.102, Z 3.100, A 0.000, B 0.000, C 0.000} C_DIS
   $VEL.CP = 0.060
   LIN  {X -9.039, Y -1.968, Z 3.100, A 0.000, B 0.000, C 0.000} C_DIS
   $VEL.CP = 0.060
   LIN  {X 1.968, Y 9.039, Z 3.100, A 0.000, B 0.000, C 0.000} C_DIS
   $VEL.CP = 0.060
   LIN  {X -1.968, Y 9.039, Z 3.100, A 0.000, B 0.000, C 0.000} C_DIS
   $VEL.CP = 0.060
   LIN  {X 7.293, Y -0.222, Z 3.100, A 0.000, B 0.000, C 0.000} C_DIS
   $VEL.CP = 0.060
   LIN  {X 7.295, Y -1.933, Z 3.100, A 0.000, B 0.000, C 0.000} C_DIS
   $VEL.CP = 0.060
   LIN  {X 9.040, Y -1.933, Z 3.100, A 0.000, B 0.000, C 0.000} C_DIS
   $VEL.CP = 0.060
   LIN  {X 9.039, Y -1.968, Z 3.100, A 0.000, B 0.000, C 0.000} C_DIS
   $VEL.CP = 0.060
   LIN  {X 9.004, Y -1.933, Z 3.100, A 0.000, B 0.000, C 0.000} C_DIS

;FOLD ARCOFF WDAT2 LIN P4 CPDAT2 Tool[1]:cmttorch Base[1]:vrashatel ;%{PE}
  ;FOLD Parameters ;%{h}
    ;Params IlfProvider=kukaroboter.arctech.arcofflin; Kuka.IsGlobalPoint=False; Kuka.PointName=P4; Kuka.BlendingEnabled=False; Kuka.MoveDataName=CPDAT2; Kuka.VelocityPath=0.01; Kuka.CurrentCDSetIndex=0; Kuka.MovementParameterFieldEnabled=True; ArcTech.WdatVarName=WDAT2; ArcTech.Basic=3.4.3.1264
  ;ENDFOLD
  $BWDSTART = FALSE
  LDAT_ACT = LCPDAT2
  FDAT_ACT = FP4
  BAS(#CP_PARAMS, gArcBasVelDefinition)
  SET_CD_PARAMS (0)
  TRIGGER WHEN PATH = ArcGetPath(#ArcOffBefore, WDAT2) DELAY = 0 DO ArcMainNG(#ArcOffBeforeOffStd, WDAT2, WP4) PRIO = -1
  TRIGGER WHEN PATH = ArcGetPath(#OnTheFlyArcOff, WDAT2) DELAY = 0 DO ArcMainNG(#ArcOffMoveStd, WDAT2, WP4) PRIO = -1
  ArcMainNG(#ArcOffBeforeMoveStd, WDAT2, WP4)
  LIN XP4
  ArcMainNG(#ArcOffAfterMoveStd, WDAT2, WP4)
;ENDFOLD
   $VEL.CP = 0.080
   LIN  {X 1.831, Y -7.480, Z 3.100, A 0.000, B 0.000, C 0.000} C_DIS
   $VEL.CP = 0.080
   LIN  {X 1.701, Y -9.040, Z 3.100, A 0.000, B 0.000, C 0.000} C_DIS

;FOLD ARCON WDAT1 LIN P3 Vel=0.5 m/s CPDAT1 Tool[1]:cmttorch Base[1]:vrashatel ;%{PE}
  ;FOLD Parameters ;%{h}
    ;Params IlfProvider=kukaroboter.arctech.arconlin; Kuka.IsGlobalPoint=False; Kuka.PointName=P3; Kuka.BlendingEnabled=False; Kuka.MoveDataName=CPDAT1; Kuka.VelocityPath=0.5; Kuka.CurrentCDSetIndex=0; Kuka.MovementParameterFieldEnabled=True; ArcTech.WdatVarName=WDAT1; ArcTech.Basic=3.4.3.1264
  ;ENDFOLD
  $BWDSTART = FALSE
  LDAT_ACT = LCPDAT1
  FDAT_ACT = FP3
  BAS(#CP_PARAMS, 0.5)
  SET_CD_PARAMS (0)
  TRIGGER WHEN DISTANCE = 1 DELAY = ArcGetDelay(#PreDefinition, WDAT1) DO ArcMainNG(#PreDefinition, WDAT1, WP3) PRIO = -1
  TRIGGER WHEN PATH = ArcGetPath(#OnTheFlyArcOn, WDAT1) DELAY = ArcGetDelay(#GasPreflow, WDAT1) DO ArcMainNG(#GasPreflow, WDAT1, WP3) PRIO = -1
  TRIGGER WHEN PATH = ArcGetPath(#OnTheFlyArcOn, WDAT1) DELAY = 0 DO ArcMainNG(#ArcOnMoveStd, WDAT1, WP3) PRIO = -1
  ArcMainNG(#ArcOnBeforeMoveStd, WDAT1, WP3)
  LIN XP3
  ArcMainNG(#ArcOnAfterMoveStd, WDAT1, WP3)
;ENDFOLD
   $VEL.CP = 0.060
   LIN  {X -2.515, Y -9.040, Z 3.100, A 0.000, B 0.000, C 0.000} C_DIS
   $VEL.CP = 0.060
   LIN  {X -2.515, Y -7.348, Z 3.100, A 0.000, B 0.000, C 0.000} C_DIS
   $VEL.CP = 0.060
   LIN  {X -5.651, Y -7.348, Z 3.100, A 0.000, B 0.000, C 0.000} C_DIS
   $VEL.CP = 0.060
   LIN  {X -5.653, Y -8.488, Z 3.100, A 0.000, B 0.000, C 0.000} C_DIS
   $VEL.CP = 0.060
   LIN  {X -9.039, Y -5.102, Z 3.100, A 0.000, B 0.000, C 0.000} C_DIS
   $VEL.CP = 0.060
   LIN  {X -9.039, Y -9.039, Z 3.100, A 0.000, B 0.000, C 0.000} C_DIS
   $VEL.CP = 0.060
   LIN  {X 9.039, Y 9.039, Z 3.100, A 0.000, B 0.000, C 0.000} C_DIS
   $VEL.CP = 0.060
   LIN  {X 5.102, Y 9.039, Z 3.100, A 0.000, B 0.000, C 0.000} C_DIS
   $VEL.CP = 0.060
   LIN  {X 9.038, Y 5.103, Z 3.100, A 0.000, B 0.000, C 0.000} C_DIS
   $VEL.CP = 0.060
   LIN  {X 9.039, Y 1.968, Z 3.100, A 0.000, B 0.000, C 0.000} C_DIS
   $VEL.CP = 0.060
   LIN  {X 8.338, Y 1.267, Z 3.100, A 0.000, B 0.000, C 0.000} C_DIS
   $VEL.CP = 0.060
   LIN  {X 7.295, Y 1.268, Z 3.100, A 0.000, B 0.000, C 0.000} C_DIS
   $VEL.CP = 0.060
   LIN  {X 7.294, Y 0.223, Z 3.100, A 0.000, B 0.000, C 0.000} C_DIS
   $VEL.CP = 0.060
   LIN  {X -1.967, Y -9.038, Z 3.100, A 0.000, B 0.000, C 0.000} C_DIS

;FOLD ARCOFF WDAT2 LIN P4 CPDAT2 Tool[1]:cmttorch Base[1]:vrashatel ;%{PE}
  ;FOLD Parameters ;%{h}
    ;Params IlfProvider=kukaroboter.arctech.arcofflin; Kuka.IsGlobalPoint=False; Kuka.PointName=P4; Kuka.BlendingEnabled=False; Kuka.MoveDataName=CPDAT2; Kuka.VelocityPath=0.01; Kuka.CurrentCDSetIndex=0; Kuka.MovementParameterFieldEnabled=True; ArcTech.WdatVarName=WDAT2; ArcTech.Basic=3.4.3.1264
  ;ENDFOLD
  $BWDSTART = FALSE
  LDAT_ACT = LCPDAT2
  FDAT_ACT = FP4
  BAS(#CP_PARAMS, gArcBasVelDefinition)
  SET_CD_PARAMS (0)
  TRIGGER WHEN PATH = ArcGetPath(#ArcOffBefore, WDAT2) DELAY = 0 DO ArcMainNG(#ArcOffBeforeOffStd, WDAT2, WP4) PRIO = -1
  TRIGGER WHEN PATH = ArcGetPath(#OnTheFlyArcOff, WDAT2) DELAY = 0 DO ArcMainNG(#ArcOffMoveStd, WDAT2, WP4) PRIO = -1
  ArcMainNG(#ArcOffBeforeMoveStd, WDAT2, WP4)
  LIN XP4
  ArcMainNG(#ArcOffAfterMoveStd, WDAT2, WP4)
;ENDFOLD
   $VEL.CP = 0.060
   LIN  {X -2.037, Y -9.108, Z 3.100, A 0.000, B 0.000, C 0.000} C_DIS
   $VEL.CP = 0.080
   LIN  {X -2.665, Y -9.010, Z 3.100, A 0.000, B 0.000, C 0.000} C_DIS

;FOLD ARCON WDAT1 LIN P3 Vel=0.5 m/s CPDAT1 Tool[1]:cmttorch Base[1]:vrashatel ;%{PE}
  ;FOLD Parameters ;%{h}
    ;Params IlfProvider=kukaroboter.arctech.arconlin; Kuka.IsGlobalPoint=False; Kuka.PointName=P3; Kuka.BlendingEnabled=False; Kuka.MoveDataName=CPDAT1; Kuka.VelocityPath=0.5; Kuka.CurrentCDSetIndex=0; Kuka.MovementParameterFieldEnabled=True; ArcTech.WdatVarName=WDAT1; ArcTech.Basic=3.4.3.1264
  ;ENDFOLD
  $BWDSTART = FALSE
  LDAT_ACT = LCPDAT1
  FDAT_ACT = FP3
  BAS(#CP_PARAMS, 0.5)
  SET_CD_PARAMS (0)
  TRIGGER WHEN DISTANCE = 1 DELAY = ArcGetDelay(#PreDefinition, WDAT1) DO ArcMainNG(#PreDefinition, WDAT1, WP3) PRIO = -1
  TRIGGER WHEN PATH = ArcGetPath(#OnTheFlyArcOn, WDAT1) DELAY = ArcGetDelay(#GasPreflow, WDAT1) DO ArcMainNG(#GasPreflow, WDAT1, WP3) PRIO = -1
  TRIGGER WHEN PATH = ArcGetPath(#OnTheFlyArcOn, WDAT1) DELAY = 0 DO ArcMainNG(#ArcOnMoveStd, WDAT1, WP3) PRIO = -1
  ArcMainNG(#ArcOnBeforeMoveStd, WDAT1, WP3)
  LIN XP3
  ArcMainNG(#ArcOnAfterMoveStd, WDAT1, WP3)
;ENDFOLD
   $VEL.CP = 0.060
   LIN  {X -2.665, Y -7.498, Z 3.100, A 0.000, B 0.000, C 0.000} C_DIS
   $VEL.CP = 0.060
   LIN  {X -5.501, Y -7.498, Z 3.100, A 0.000, B 0.000, C 0.000} C_DIS
   $VEL.CP = 0.060
   LIN  {X -5.503, Y -9.010, Z 3.100, A 0.000, B 0.000, C 0.000} C_DIS
   $VEL.CP = 0.060
   LIN  {X -2.665, Y -9.010, Z 3.100, A 0.000, B 0.000, C 0.000} C_DIS

;FOLD ARCOFF WDAT2 LIN P4 CPDAT2 Tool[1]:cmttorch Base[1]:vrashatel ;%{PE}
  ;FOLD Parameters ;%{h}
    ;Params IlfProvider=kukaroboter.arctech.arcofflin; Kuka.IsGlobalPoint=False; Kuka.PointName=P4; Kuka.BlendingEnabled=False; Kuka.MoveDataName=CPDAT2; Kuka.VelocityPath=0.01; Kuka.CurrentCDSetIndex=0; Kuka.MovementParameterFieldEnabled=True; ArcTech.WdatVarName=WDAT2; ArcTech.Basic=3.4.3.1264
  ;ENDFOLD
  $BWDSTART = FALSE
  LDAT_ACT = LCPDAT2
  FDAT_ACT = FP4
  BAS(#CP_PARAMS, gArcBasVelDefinition)
  SET_CD_PARAMS (0)
  TRIGGER WHEN PATH = ArcGetPath(#ArcOffBefore, WDAT2) DELAY = 0 DO ArcMainNG(#ArcOffBeforeOffStd, WDAT2, WP4) PRIO = -1
  TRIGGER WHEN PATH = ArcGetPath(#OnTheFlyArcOff, WDAT2) DELAY = 0 DO ArcMainNG(#ArcOffMoveStd, WDAT2, WP4) PRIO = -1
  ArcMainNG(#ArcOffBeforeMoveStd, WDAT2, WP4)
  LIN XP4
  ArcMainNG(#ArcOffAfterMoveStd, WDAT2, WP4)
;ENDFOLD
   $VEL.CP = 0.080
   LIN  {X -3.172, Y -8.828, Z 3.100, A 0.000, B 0.000, C 0.000} C_DIS

;FOLD ARCON WDAT1 LIN P3 Vel=0.5 m/s CPDAT1 Tool[1]:cmttorch Base[1]:vrashatel ;%{PE}
  ;FOLD Parameters ;%{h}
    ;Params IlfProvider=kukaroboter.arctech.arconlin; Kuka.IsGlobalPoint=False; Kuka.PointName=P3; Kuka.BlendingEnabled=False; Kuka.MoveDataName=CPDAT1; Kuka.VelocityPath=0.5; Kuka.CurrentCDSetIndex=0; Kuka.MovementParameterFieldEnabled=True; ArcTech.WdatVarName=WDAT1; ArcTech.Basic=3.4.3.1264
  ;ENDFOLD
  $BWDSTART = FALSE
  LDAT_ACT = LCPDAT1
  FDAT_ACT = FP3
  BAS(#CP_PARAMS, 0.5)
  SET_CD_PARAMS (0)
  TRIGGER WHEN DISTANCE = 1 DELAY = ArcGetDelay(#PreDefinition, WDAT1) DO ArcMainNG(#PreDefinition, WDAT1, WP3) PRIO = -1
  TRIGGER WHEN PATH = ArcGetPath(#OnTheFlyArcOn, WDAT1) DELAY = ArcGetDelay(#GasPreflow, WDAT1) DO ArcMainNG(#GasPreflow, WDAT1, WP3) PRIO = -1
  TRIGGER WHEN PATH = ArcGetPath(#OnTheFlyArcOn, WDAT1) DELAY = 0 DO ArcMainNG(#ArcOnMoveStd, WDAT1, WP3) PRIO = -1
  ArcMainNG(#ArcOnBeforeMoveStd, WDAT1, WP3)
  LIN XP3
  ArcMainNG(#ArcOnAfterMoveStd, WDAT1, WP3)
;ENDFOLD
   $VEL.CP = 0.060
   LIN  {X -2.844, Y -8.501, Z 3.100, A 0.000, B 0.000, C 0.000} C_DIS

;FOLD ARCOFF WDAT2 LIN P4 CPDAT2 Tool[1]:cmttorch Base[1]:vrashatel ;%{PE}
  ;FOLD Parameters ;%{h}
    ;Params IlfProvider=kukaroboter.arctech.arcofflin; Kuka.IsGlobalPoint=False; Kuka.PointName=P4; Kuka.BlendingEnabled=False; Kuka.MoveDataName=CPDAT2; Kuka.VelocityPath=0.01; Kuka.CurrentCDSetIndex=0; Kuka.MovementParameterFieldEnabled=True; ArcTech.WdatVarName=WDAT2; ArcTech.Basic=3.4.3.1264
  ;ENDFOLD
  $BWDSTART = FALSE
  LDAT_ACT = LCPDAT2
  FDAT_ACT = FP4
  BAS(#CP_PARAMS, gArcBasVelDefinition)
  SET_CD_PARAMS (0)
  TRIGGER WHEN PATH = ArcGetPath(#ArcOffBefore, WDAT2) DELAY = 0 DO ArcMainNG(#ArcOffBeforeOffStd, WDAT2, WP4) PRIO = -1
  TRIGGER WHEN PATH = ArcGetPath(#OnTheFlyArcOff, WDAT2) DELAY = 0 DO ArcMainNG(#ArcOffMoveStd, WDAT2, WP4) PRIO = -1
  ArcMainNG(#ArcOffBeforeMoveStd, WDAT2, WP4)
  LIN XP4
  ArcMainNG(#ArcOffAfterMoveStd, WDAT2, WP4)
;ENDFOLD
   $VEL.CP = 0.080
   LIN  {X -2.844, Y -7.935, Z 3.100, A 0.000, B 0.000, C 0.000} C_DIS

;FOLD ARCON WDAT1 LIN P3 Vel=0.5 m/s CPDAT1 Tool[1]:cmttorch Base[1]:vrashatel ;%{PE}
  ;FOLD Parameters ;%{h}
    ;Params IlfProvider=kukaroboter.arctech.arconlin; Kuka.IsGlobalPoint=False; Kuka.PointName=P3; Kuka.BlendingEnabled=False; Kuka.MoveDataName=CPDAT1; Kuka.VelocityPath=0.5; Kuka.CurrentCDSetIndex=0; Kuka.MovementParameterFieldEnabled=True; ArcTech.WdatVarName=WDAT1; ArcTech.Basic=3.4.3.1264
  ;ENDFOLD
  $BWDSTART = FALSE
  LDAT_ACT = LCPDAT1
  FDAT_ACT = FP3
  BAS(#CP_PARAMS, 0.5)
  SET_CD_PARAMS (0)
  TRIGGER WHEN DISTANCE = 1 DELAY = ArcGetDelay(#PreDefinition, WDAT1) DO ArcMainNG(#PreDefinition, WDAT1, WP3) PRIO = -1
  TRIGGER WHEN PATH = ArcGetPath(#OnTheFlyArcOn, WDAT1) DELAY = ArcGetDelay(#GasPreflow, WDAT1) DO ArcMainNG(#GasPreflow, WDAT1, WP3) PRIO = -1
  TRIGGER WHEN PATH = ArcGetPath(#OnTheFlyArcOn, WDAT1) DELAY = 0 DO ArcMainNG(#ArcOnMoveStd, WDAT1, WP3) PRIO = -1
  ArcMainNG(#ArcOnBeforeMoveStd, WDAT1, WP3)
  LIN XP3
  ArcMainNG(#ArcOnAfterMoveStd, WDAT1, WP3)
;ENDFOLD
   $VEL.CP = 0.060
   LIN  {X -3.737, Y -8.828, Z 3.100, A 0.000, B 0.000, C 0.000} C_DIS

;FOLD ARCOFF WDAT2 LIN P4 CPDAT2 Tool[1]:cmttorch Base[1]:vrashatel ;%{PE}
  ;FOLD Parameters ;%{h}
    ;Params IlfProvider=kukaroboter.arctech.arcofflin; Kuka.IsGlobalPoint=False; Kuka.PointName=P4; Kuka.BlendingEnabled=False; Kuka.MoveDataName=CPDAT2; Kuka.VelocityPath=0.01; Kuka.CurrentCDSetIndex=0; Kuka.MovementParameterFieldEnabled=True; ArcTech.WdatVarName=WDAT2; ArcTech.Basic=3.4.3.1264
  ;ENDFOLD
  $BWDSTART = FALSE
  LDAT_ACT = LCPDAT2
  FDAT_ACT = FP4
  BAS(#CP_PARAMS, gArcBasVelDefinition)
  SET_CD_PARAMS (0)
  TRIGGER WHEN PATH = ArcGetPath(#ArcOffBefore, WDAT2) DELAY = 0 DO ArcMainNG(#ArcOffBeforeOffStd, WDAT2, WP4) PRIO = -1
  TRIGGER WHEN PATH = ArcGetPath(#OnTheFlyArcOff, WDAT2) DELAY = 0 DO ArcMainNG(#ArcOffMoveStd, WDAT2, WP4) PRIO = -1
  ArcMainNG(#ArcOffBeforeMoveStd, WDAT2, WP4)
  LIN XP4
  ArcMainNG(#ArcOffAfterMoveStd, WDAT2, WP4)
;ENDFOLD
   $VEL.CP = 0.080
   LIN  {X -4.303, Y -8.828, Z 3.100, A 0.000, B 0.000, C 0.000} C_DIS

;FOLD ARCON WDAT1 LIN P3 Vel=0.5 m/s CPDAT1 Tool[1]:cmttorch Base[1]:vrashatel ;%{PE}
  ;FOLD Parameters ;%{h}
    ;Params IlfProvider=kukaroboter.arctech.arconlin; Kuka.IsGlobalPoint=False; Kuka.PointName=P3; Kuka.BlendingEnabled=False; Kuka.MoveDataName=CPDAT1; Kuka.VelocityPath=0.5; Kuka.CurrentCDSetIndex=0; Kuka.MovementParameterFieldEnabled=True; ArcTech.WdatVarName=WDAT1; ArcTech.Basic=3.4.3.1264
  ;ENDFOLD
  $BWDSTART = FALSE
  LDAT_ACT = LCPDAT1
  FDAT_ACT = FP3
  BAS(#CP_PARAMS, 0.5)
  SET_CD_PARAMS (0)
  TRIGGER WHEN DISTANCE = 1 DELAY = ArcGetDelay(#PreDefinition, WDAT1) DO ArcMainNG(#PreDefinition, WDAT1, WP3) PRIO = -1
  TRIGGER WHEN PATH = ArcGetPath(#OnTheFlyArcOn, WDAT1) DELAY = ArcGetDelay(#GasPreflow, WDAT1) DO ArcMainNG(#GasPreflow, WDAT1, WP3) PRIO = -1
  TRIGGER WHEN PATH = ArcGetPath(#OnTheFlyArcOn, WDAT1) DELAY = 0 DO ArcMainNG(#ArcOnMoveStd, WDAT1, WP3) PRIO = -1
  ArcMainNG(#ArcOnBeforeMoveStd, WDAT1, WP3)
  LIN XP3
  ArcMainNG(#ArcOnAfterMoveStd, WDAT1, WP3)
;ENDFOLD
   $VEL.CP = 0.060
   LIN  {X -3.151, Y -7.677, Z 3.100, A 0.000, B 0.000, C 0.000} C_DIS

;FOLD ARCOFF WDAT2 LIN P4 CPDAT2 Tool[1]:cmttorch Base[1]:vrashatel ;%{PE}
  ;FOLD Parameters ;%{h}
    ;Params IlfProvider=kukaroboter.arctech.arcofflin; Kuka.IsGlobalPoint=False; Kuka.PointName=P4; Kuka.BlendingEnabled=False; Kuka.MoveDataName=CPDAT2; Kuka.VelocityPath=0.01; Kuka.CurrentCDSetIndex=0; Kuka.MovementParameterFieldEnabled=True; ArcTech.WdatVarName=WDAT2; ArcTech.Basic=3.4.3.1264
  ;ENDFOLD
  $BWDSTART = FALSE
  LDAT_ACT = LCPDAT2
  FDAT_ACT = FP4
  BAS(#CP_PARAMS, gArcBasVelDefinition)
  SET_CD_PARAMS (0)
  TRIGGER WHEN PATH = ArcGetPath(#ArcOffBefore, WDAT2) DELAY = 0 DO ArcMainNG(#ArcOffBeforeOffStd, WDAT2, WP4) PRIO = -1
  TRIGGER WHEN PATH = ArcGetPath(#OnTheFlyArcOff, WDAT2) DELAY = 0 DO ArcMainNG(#ArcOffMoveStd, WDAT2, WP4) PRIO = -1
  ArcMainNG(#ArcOffBeforeMoveStd, WDAT2, WP4)
  LIN XP4
  ArcMainNG(#ArcOffAfterMoveStd, WDAT2, WP4)
;ENDFOLD
   $VEL.CP = 0.080
   LIN  {X -3.717, Y -7.677, Z 3.100, A 0.000, B 0.000, C 0.000} C_DIS

;FOLD ARCON WDAT1 LIN P3 Vel=0.5 m/s CPDAT1 Tool[1]:cmttorch Base[1]:vrashatel ;%{PE}
  ;FOLD Parameters ;%{h}
    ;Params IlfProvider=kukaroboter.arctech.arconlin; Kuka.IsGlobalPoint=False; Kuka.PointName=P3; Kuka.BlendingEnabled=False; Kuka.MoveDataName=CPDAT1; Kuka.VelocityPath=0.5; Kuka.CurrentCDSetIndex=0; Kuka.MovementParameterFieldEnabled=True; ArcTech.WdatVarName=WDAT1; ArcTech.Basic=3.4.3.1264
  ;ENDFOLD
  $BWDSTART = FALSE
  LDAT_ACT = LCPDAT1
  FDAT_ACT = FP3
  BAS(#CP_PARAMS, 0.5)
  SET_CD_PARAMS (0)
  TRIGGER WHEN DISTANCE = 1 DELAY = ArcGetDelay(#PreDefinition, WDAT1) DO ArcMainNG(#PreDefinition, WDAT1, WP3) PRIO = -1
  TRIGGER WHEN PATH = ArcGetPath(#OnTheFlyArcOn, WDAT1) DELAY = ArcGetDelay(#GasPreflow, WDAT1) DO ArcMainNG(#GasPreflow, WDAT1, WP3) PRIO = -1
  TRIGGER WHEN PATH = ArcGetPath(#OnTheFlyArcOn, WDAT1) DELAY = 0 DO ArcMainNG(#ArcOnMoveStd, WDAT1, WP3) PRIO = -1
  ArcMainNG(#ArcOnBeforeMoveStd, WDAT1, WP3)
  LIN XP3
  ArcMainNG(#ArcOnAfterMoveStd, WDAT1, WP3)
;ENDFOLD
   $VEL.CP = 0.060
   LIN  {X -4.869, Y -8.828, Z 3.100, A 0.000, B 0.000, C 0.000} C_DIS

;FOLD ARCOFF WDAT2 LIN P4 CPDAT2 Tool[1]:cmttorch Base[1]:vrashatel ;%{PE}
  ;FOLD Parameters ;%{h}
    ;Params IlfProvider=kukaroboter.arctech.arcofflin; Kuka.IsGlobalPoint=False; Kuka.PointName=P4; Kuka.BlendingEnabled=False; Kuka.MoveDataName=CPDAT2; Kuka.VelocityPath=0.01; Kuka.CurrentCDSetIndex=0; Kuka.MovementParameterFieldEnabled=True; ArcTech.WdatVarName=WDAT2; ArcTech.Basic=3.4.3.1264
  ;ENDFOLD
  $BWDSTART = FALSE
  LDAT_ACT = LCPDAT2
  FDAT_ACT = FP4
  BAS(#CP_PARAMS, gArcBasVelDefinition)
  SET_CD_PARAMS (0)
  TRIGGER WHEN PATH = ArcGetPath(#ArcOffBefore, WDAT2) DELAY = 0 DO ArcMainNG(#ArcOffBeforeOffStd, WDAT2, WP4) PRIO = -1
  TRIGGER WHEN PATH = ArcGetPath(#OnTheFlyArcOff, WDAT2) DELAY = 0 DO ArcMainNG(#ArcOffMoveStd, WDAT2, WP4) PRIO = -1
  ArcMainNG(#ArcOffBeforeMoveStd, WDAT2, WP4)
  LIN XP4
  ArcMainNG(#ArcOffAfterMoveStd, WDAT2, WP4)
;ENDFOLD
   $VEL.CP = 0.080
   LIN  {X -5.323, Y -8.717, Z 3.100, A 0.000, B 0.000, C 0.000} C_DIS

;FOLD ARCON WDAT1 LIN P3 Vel=0.5 m/s CPDAT1 Tool[1]:cmttorch Base[1]:vrashatel ;%{PE}
  ;FOLD Parameters ;%{h}
    ;Params IlfProvider=kukaroboter.arctech.arconlin; Kuka.IsGlobalPoint=False; Kuka.PointName=P3; Kuka.BlendingEnabled=False; Kuka.MoveDataName=CPDAT1; Kuka.VelocityPath=0.5; Kuka.CurrentCDSetIndex=0; Kuka.MovementParameterFieldEnabled=True; ArcTech.WdatVarName=WDAT1; ArcTech.Basic=3.4.3.1264
  ;ENDFOLD
  $BWDSTART = FALSE
  LDAT_ACT = LCPDAT1
  FDAT_ACT = FP3
  BAS(#CP_PARAMS, 0.5)
  SET_CD_PARAMS (0)
  TRIGGER WHEN DISTANCE = 1 DELAY = ArcGetDelay(#PreDefinition, WDAT1) DO ArcMainNG(#PreDefinition, WDAT1, WP3) PRIO = -1
  TRIGGER WHEN PATH = ArcGetPath(#OnTheFlyArcOn, WDAT1) DELAY = ArcGetDelay(#GasPreflow, WDAT1) DO ArcMainNG(#GasPreflow, WDAT1, WP3) PRIO = -1
  TRIGGER WHEN PATH = ArcGetPath(#OnTheFlyArcOn, WDAT1) DELAY = 0 DO ArcMainNG(#ArcOnMoveStd, WDAT1, WP3) PRIO = -1
  ArcMainNG(#ArcOnBeforeMoveStd, WDAT1, WP3)
  LIN XP3
  ArcMainNG(#ArcOnAfterMoveStd, WDAT1, WP3)
;ENDFOLD
   $VEL.CP = 0.060
   LIN  {X -4.282, Y -7.677, Z 3.100, A 0.000, B 0.000, C 0.000} C_DIS

;FOLD ARCOFF WDAT2 LIN P4 CPDAT2 Tool[1]:cmttorch Base[1]:vrashatel ;%{PE}
  ;FOLD Parameters ;%{h}
    ;Params IlfProvider=kukaroboter.arctech.arcofflin; Kuka.IsGlobalPoint=False; Kuka.PointName=P4; Kuka.BlendingEnabled=False; Kuka.MoveDataName=CPDAT2; Kuka.VelocityPath=0.01; Kuka.CurrentCDSetIndex=0; Kuka.MovementParameterFieldEnabled=True; ArcTech.WdatVarName=WDAT2; ArcTech.Basic=3.4.3.1264
  ;ENDFOLD
  $BWDSTART = FALSE
  LDAT_ACT = LCPDAT2
  FDAT_ACT = FP4
  BAS(#CP_PARAMS, gArcBasVelDefinition)
  SET_CD_PARAMS (0)
  TRIGGER WHEN PATH = ArcGetPath(#ArcOffBefore, WDAT2) DELAY = 0 DO ArcMainNG(#ArcOffBeforeOffStd, WDAT2, WP4) PRIO = -1
  TRIGGER WHEN PATH = ArcGetPath(#OnTheFlyArcOff, WDAT2) DELAY = 0 DO ArcMainNG(#ArcOffMoveStd, WDAT2, WP4) PRIO = -1
  ArcMainNG(#ArcOffBeforeMoveStd, WDAT2, WP4)
  LIN XP4
  ArcMainNG(#ArcOffAfterMoveStd, WDAT2, WP4)
;ENDFOLD
   $VEL.CP = 0.080
   LIN  {X -4.848, Y -7.677, Z 3.100, A 0.000, B 0.000, C 0.000} C_DIS

;FOLD ARCON WDAT1 LIN P3 Vel=0.5 m/s CPDAT1 Tool[1]:cmttorch Base[1]:vrashatel ;%{PE}
  ;FOLD Parameters ;%{h}
    ;Params IlfProvider=kukaroboter.arctech.arconlin; Kuka.IsGlobalPoint=False; Kuka.PointName=P3; Kuka.BlendingEnabled=False; Kuka.MoveDataName=CPDAT1; Kuka.VelocityPath=0.5; Kuka.CurrentCDSetIndex=0; Kuka.MovementParameterFieldEnabled=True; ArcTech.WdatVarName=WDAT1; ArcTech.Basic=3.4.3.1264
  ;ENDFOLD
  $BWDSTART = FALSE
  LDAT_ACT = LCPDAT1
  FDAT_ACT = FP3
  BAS(#CP_PARAMS, 0.5)
  SET_CD_PARAMS (0)
  TRIGGER WHEN DISTANCE = 1 DELAY = ArcGetDelay(#PreDefinition, WDAT1) DO ArcMainNG(#PreDefinition, WDAT1, WP3) PRIO = -1
  TRIGGER WHEN PATH = ArcGetPath(#OnTheFlyArcOn, WDAT1) DELAY = ArcGetDelay(#GasPreflow, WDAT1) DO ArcMainNG(#GasPreflow, WDAT1, WP3) PRIO = -1
  TRIGGER WHEN PATH = ArcGetPath(#OnTheFlyArcOn, WDAT1) DELAY = 0 DO ArcMainNG(#ArcOnMoveStd, WDAT1, WP3) PRIO = -1
  ArcMainNG(#ArcOnBeforeMoveStd, WDAT1, WP3)
  LIN XP3
  ArcMainNG(#ArcOnAfterMoveStd, WDAT1, WP3)
;ENDFOLD
   $VEL.CP = 0.060
   LIN  {X -5.322, Y -8.150, Z 3.100, A 0.000, B 0.000, C 0.000} C_DIS

;FOLD ARCOFF WDAT2 LIN P4 CPDAT2 Tool[1]:cmttorch Base[1]:vrashatel ;%{PE}
  ;FOLD Parameters ;%{h}
    ;Params IlfProvider=kukaroboter.arctech.arcofflin; Kuka.IsGlobalPoint=False; Kuka.PointName=P4; Kuka.BlendingEnabled=False; Kuka.MoveDataName=CPDAT2; Kuka.VelocityPath=0.01; Kuka.CurrentCDSetIndex=0; Kuka.MovementParameterFieldEnabled=True; ArcTech.WdatVarName=WDAT2; ArcTech.Basic=3.4.3.1264
  ;ENDFOLD
  $BWDSTART = FALSE
  LDAT_ACT = LCPDAT2
  FDAT_ACT = FP4
  BAS(#CP_PARAMS, gArcBasVelDefinition)
  SET_CD_PARAMS (0)
  TRIGGER WHEN PATH = ArcGetPath(#ArcOffBefore, WDAT2) DELAY = 0 DO ArcMainNG(#ArcOffBeforeOffStd, WDAT2, WP4) PRIO = -1
  TRIGGER WHEN PATH = ArcGetPath(#OnTheFlyArcOff, WDAT2) DELAY = 0 DO ArcMainNG(#ArcOffMoveStd, WDAT2, WP4) PRIO = -1
  ArcMainNG(#ArcOffBeforeMoveStd, WDAT2, WP4)
  LIN XP4
  ArcMainNG(#ArcOffAfterMoveStd, WDAT2, WP4)
;ENDFOLD
   $VEL.CP = 0.080
   LIN  {X -5.592, Y -8.150, Z 3.100, A 0.000, B 0.000, C 0.000} C_DIS
   $VEL.CP = 0.080
   LIN  {X -5.519, Y -7.480, Z 3.100, A 0.000, B 0.000, C 0.000} C_DIS
   $VEL.CP = 0.080
   LIN  {X 1.789, Y -7.438, Z 3.100, A 0.000, B 0.000, C 0.000} C_DIS
   $VEL.CP = 0.080
   LIN  {X 1.849, Y -7.498, Z 3.100, A 0.000, B 0.000, C 0.000} C_DIS

;FOLD ARCON WDAT1 LIN P3 Vel=0.5 m/s CPDAT1 Tool[1]:cmttorch Base[1]:vrashatel ;%{PE}
  ;FOLD Parameters ;%{h}
    ;Params IlfProvider=kukaroboter.arctech.arconlin; Kuka.IsGlobalPoint=False; Kuka.PointName=P3; Kuka.BlendingEnabled=False; Kuka.MoveDataName=CPDAT1; Kuka.VelocityPath=0.5; Kuka.CurrentCDSetIndex=0; Kuka.MovementParameterFieldEnabled=True; ArcTech.WdatVarName=WDAT1; ArcTech.Basic=3.4.3.1264
  ;ENDFOLD
  $BWDSTART = FALSE
  LDAT_ACT = LCPDAT1
  FDAT_ACT = FP3
  BAS(#CP_PARAMS, 0.5)
  SET_CD_PARAMS (0)
  TRIGGER WHEN DISTANCE = 1 DELAY = ArcGetDelay(#PreDefinition, WDAT1) DO ArcMainNG(#PreDefinition, WDAT1, WP3) PRIO = -1
  TRIGGER WHEN PATH = ArcGetPath(#OnTheFlyArcOn, WDAT1) DELAY = ArcGetDelay(#GasPreflow, WDAT1) DO ArcMainNG(#GasPreflow, WDAT1, WP3) PRIO = -1
  TRIGGER WHEN PATH = ArcGetPath(#OnTheFlyArcOn, WDAT1) DELAY = 0 DO ArcMainNG(#ArcOnMoveStd, WDAT1, WP3) PRIO = -1
  ArcMainNG(#ArcOnBeforeMoveStd, WDAT1, WP3)
  LIN XP3
  ArcMainNG(#ArcOnAfterMoveStd, WDAT1, WP3)
;ENDFOLD
   $VEL.CP = 0.060
   LIN  {X 1.851, Y -9.010, Z 3.100, A 0.000, B 0.000, C 0.000} C_DIS
   $VEL.CP = 0.060
   LIN  {X 4.850, Y -9.010, Z 3.100, A 0.000, B 0.000, C 0.000} C_DIS
   $VEL.CP = 0.060
   LIN  {X 4.848, Y -7.498, Z 3.100, A 0.000, B 0.000, C 0.000} C_DIS
   $VEL.CP = 0.060
   LIN  {X 1.849, Y -7.498, Z 3.100, A 0.000, B 0.000, C 0.000} C_DIS

;FOLD ARCOFF WDAT2 LIN P4 CPDAT2 Tool[1]:cmttorch Base[1]:vrashatel ;%{PE}
  ;FOLD Parameters ;%{h}
    ;Params IlfProvider=kukaroboter.arctech.arcofflin; Kuka.IsGlobalPoint=False; Kuka.PointName=P4; Kuka.BlendingEnabled=False; Kuka.MoveDataName=CPDAT2; Kuka.VelocityPath=0.01; Kuka.CurrentCDSetIndex=0; Kuka.MovementParameterFieldEnabled=True; ArcTech.WdatVarName=WDAT2; ArcTech.Basic=3.4.3.1264
  ;ENDFOLD
  $BWDSTART = FALSE
  LDAT_ACT = LCPDAT2
  FDAT_ACT = FP4
  BAS(#CP_PARAMS, gArcBasVelDefinition)
  SET_CD_PARAMS (0)
  TRIGGER WHEN PATH = ArcGetPath(#ArcOffBefore, WDAT2) DELAY = 0 DO ArcMainNG(#ArcOffBeforeOffStd, WDAT2, WP4) PRIO = -1
  TRIGGER WHEN PATH = ArcGetPath(#OnTheFlyArcOff, WDAT2) DELAY = 0 DO ArcMainNG(#ArcOffMoveStd, WDAT2, WP4) PRIO = -1
  ArcMainNG(#ArcOffBeforeMoveStd, WDAT2, WP4)
  LIN XP4
  ArcMainNG(#ArcOffAfterMoveStd, WDAT2, WP4)
;ENDFOLD
   $VEL.CP = 0.080
   LIN  {X 2.029, Y -8.152, Z 3.100, A 0.000, B 0.000, C 0.000} C_DIS

;FOLD ARCON WDAT1 LIN P3 Vel=0.5 m/s CPDAT1 Tool[1]:cmttorch Base[1]:vrashatel ;%{PE}
  ;FOLD Parameters ;%{h}
    ;Params IlfProvider=kukaroboter.arctech.arconlin; Kuka.IsGlobalPoint=False; Kuka.PointName=P3; Kuka.BlendingEnabled=False; Kuka.MoveDataName=CPDAT1; Kuka.VelocityPath=0.5; Kuka.CurrentCDSetIndex=0; Kuka.MovementParameterFieldEnabled=True; ArcTech.WdatVarName=WDAT1; ArcTech.Basic=3.4.3.1264
  ;ENDFOLD
  $BWDSTART = FALSE
  LDAT_ACT = LCPDAT1
  FDAT_ACT = FP3
  BAS(#CP_PARAMS, 0.5)
  SET_CD_PARAMS (0)
  TRIGGER WHEN DISTANCE = 1 DELAY = ArcGetDelay(#PreDefinition, WDAT1) DO ArcMainNG(#PreDefinition, WDAT1, WP3) PRIO = -1
  TRIGGER WHEN PATH = ArcGetPath(#OnTheFlyArcOn, WDAT1) DELAY = ArcGetDelay(#GasPreflow, WDAT1) DO ArcMainNG(#GasPreflow, WDAT1, WP3) PRIO = -1
  TRIGGER WHEN PATH = ArcGetPath(#OnTheFlyArcOn, WDAT1) DELAY = 0 DO ArcMainNG(#ArcOnMoveStd, WDAT1, WP3) PRIO = -1
  ArcMainNG(#ArcOnBeforeMoveStd, WDAT1, WP3)
  LIN XP3
  ArcMainNG(#ArcOnAfterMoveStd, WDAT1, WP3)
;ENDFOLD
   $VEL.CP = 0.060
   LIN  {X 2.505, Y -7.677, Z 3.100, A 0.000, B 0.000, C 0.000} C_DIS

;FOLD ARCOFF WDAT2 LIN P4 CPDAT2 Tool[1]:cmttorch Base[1]:vrashatel ;%{PE}
  ;FOLD Parameters ;%{h}
    ;Params IlfProvider=kukaroboter.arctech.arcofflin; Kuka.IsGlobalPoint=False; Kuka.PointName=P4; Kuka.BlendingEnabled=False; Kuka.MoveDataName=CPDAT2; Kuka.VelocityPath=0.01; Kuka.CurrentCDSetIndex=0; Kuka.MovementParameterFieldEnabled=True; ArcTech.WdatVarName=WDAT2; ArcTech.Basic=3.4.3.1264
  ;ENDFOLD
  $BWDSTART = FALSE
  LDAT_ACT = LCPDAT2
  FDAT_ACT = FP4
  BAS(#CP_PARAMS, gArcBasVelDefinition)
  SET_CD_PARAMS (0)
  TRIGGER WHEN PATH = ArcGetPath(#ArcOffBefore, WDAT2) DELAY = 0 DO ArcMainNG(#ArcOffBeforeOffStd, WDAT2, WP4) PRIO = -1
  TRIGGER WHEN PATH = ArcGetPath(#OnTheFlyArcOff, WDAT2) DELAY = 0 DO ArcMainNG(#ArcOffMoveStd, WDAT2, WP4) PRIO = -1
  ArcMainNG(#ArcOffBeforeMoveStd, WDAT2, WP4)
  LIN XP4
  ArcMainNG(#ArcOffAfterMoveStd, WDAT2, WP4)
;ENDFOLD
   $VEL.CP = 0.080
   LIN  {X 3.070, Y -7.677, Z 3.100, A 0.000, B 0.000, C 0.000} C_DIS

;FOLD ARCON WDAT1 LIN P3 Vel=0.5 m/s CPDAT1 Tool[1]:cmttorch Base[1]:vrashatel ;%{PE}
  ;FOLD Parameters ;%{h}
    ;Params IlfProvider=kukaroboter.arctech.arconlin; Kuka.IsGlobalPoint=False; Kuka.PointName=P3; Kuka.BlendingEnabled=False; Kuka.MoveDataName=CPDAT1; Kuka.VelocityPath=0.5; Kuka.CurrentCDSetIndex=0; Kuka.MovementParameterFieldEnabled=True; ArcTech.WdatVarName=WDAT1; ArcTech.Basic=3.4.3.1264
  ;ENDFOLD
  $BWDSTART = FALSE
  LDAT_ACT = LCPDAT1
  FDAT_ACT = FP3
  BAS(#CP_PARAMS, 0.5)
  SET_CD_PARAMS (0)
  TRIGGER WHEN DISTANCE = 1 DELAY = ArcGetDelay(#PreDefinition, WDAT1) DO ArcMainNG(#PreDefinition, WDAT1, WP3) PRIO = -1
  TRIGGER WHEN PATH = ArcGetPath(#OnTheFlyArcOn, WDAT1) DELAY = ArcGetDelay(#GasPreflow, WDAT1) DO ArcMainNG(#GasPreflow, WDAT1, WP3) PRIO = -1
  TRIGGER WHEN PATH = ArcGetPath(#OnTheFlyArcOn, WDAT1) DELAY = 0 DO ArcMainNG(#ArcOnMoveStd, WDAT1, WP3) PRIO = -1
  ArcMainNG(#ArcOnBeforeMoveStd, WDAT1, WP3)
  LIN XP3
  ArcMainNG(#ArcOnAfterMoveStd, WDAT1, WP3)
;ENDFOLD
   $VEL.CP = 0.060
   LIN  {X 2.030, Y -8.717, Z 3.100, A 0.000, B 0.000, C 0.000} C_DIS

;FOLD ARCOFF WDAT2 LIN P4 CPDAT2 Tool[1]:cmttorch Base[1]:vrashatel ;%{PE}
  ;FOLD Parameters ;%{h}
    ;Params IlfProvider=kukaroboter.arctech.arcofflin; Kuka.IsGlobalPoint=False; Kuka.PointName=P4; Kuka.BlendingEnabled=False; Kuka.MoveDataName=CPDAT2; Kuka.VelocityPath=0.01; Kuka.CurrentCDSetIndex=0; Kuka.MovementParameterFieldEnabled=True; ArcTech.WdatVarName=WDAT2; ArcTech.Basic=3.4.3.1264
  ;ENDFOLD
  $BWDSTART = FALSE
  LDAT_ACT = LCPDAT2
  FDAT_ACT = FP4
  BAS(#CP_PARAMS, gArcBasVelDefinition)
  SET_CD_PARAMS (0)
  TRIGGER WHEN PATH = ArcGetPath(#ArcOffBefore, WDAT2) DELAY = 0 DO ArcMainNG(#ArcOffBeforeOffStd, WDAT2, WP4) PRIO = -1
  TRIGGER WHEN PATH = ArcGetPath(#OnTheFlyArcOff, WDAT2) DELAY = 0 DO ArcMainNG(#ArcOffMoveStd, WDAT2, WP4) PRIO = -1
  ArcMainNG(#ArcOffBeforeMoveStd, WDAT2, WP4)
  LIN XP4
  ArcMainNG(#ArcOffAfterMoveStd, WDAT2, WP4)
;ENDFOLD
   $VEL.CP = 0.080
   LIN  {X 2.484, Y -8.828, Z 3.100, A 0.000, B 0.000, C 0.000} C_DIS

;FOLD ARCON WDAT1 LIN P3 Vel=0.5 m/s CPDAT1 Tool[1]:cmttorch Base[1]:vrashatel ;%{PE}
  ;FOLD Parameters ;%{h}
    ;Params IlfProvider=kukaroboter.arctech.arconlin; Kuka.IsGlobalPoint=False; Kuka.PointName=P3; Kuka.BlendingEnabled=False; Kuka.MoveDataName=CPDAT1; Kuka.VelocityPath=0.5; Kuka.CurrentCDSetIndex=0; Kuka.MovementParameterFieldEnabled=True; ArcTech.WdatVarName=WDAT1; ArcTech.Basic=3.4.3.1264
  ;ENDFOLD
  $BWDSTART = FALSE
  LDAT_ACT = LCPDAT1
  FDAT_ACT = FP3
  BAS(#CP_PARAMS, 0.5)
  SET_CD_PARAMS (0)
  TRIGGER WHEN DISTANCE = 1 DELAY = ArcGetDelay(#PreDefinition, WDAT1) DO ArcMainNG(#PreDefinition, WDAT1, WP3) PRIO = -1
  TRIGGER WHEN PATH = ArcGetPath(#OnTheFlyArcOn, WDAT1) DELAY = ArcGetDelay(#GasPreflow, WDAT1) DO ArcMainNG(#GasPreflow, WDAT1, WP3) PRIO = -1
  TRIGGER WHEN PATH = ArcGetPath(#OnTheFlyArcOn, WDAT1) DELAY = 0 DO ArcMainNG(#ArcOnMoveStd, WDAT1, WP3) PRIO = -1
  ArcMainNG(#ArcOnBeforeMoveStd, WDAT1, WP3)
  LIN XP3
  ArcMainNG(#ArcOnAfterMoveStd, WDAT1, WP3)
;ENDFOLD
   $VEL.CP = 0.060
   LIN  {X 3.636, Y -7.677, Z 3.100, A 0.000, B 0.000, C 0.000} C_DIS

;FOLD ARCOFF WDAT2 LIN P4 CPDAT2 Tool[1]:cmttorch Base[1]:vrashatel ;%{PE}
  ;FOLD Parameters ;%{h}
    ;Params IlfProvider=kukaroboter.arctech.arcofflin; Kuka.IsGlobalPoint=False; Kuka.PointName=P4; Kuka.BlendingEnabled=False; Kuka.MoveDataName=CPDAT2; Kuka.VelocityPath=0.01; Kuka.CurrentCDSetIndex=0; Kuka.MovementParameterFieldEnabled=True; ArcTech.WdatVarName=WDAT2; ArcTech.Basic=3.4.3.1264
  ;ENDFOLD
  $BWDSTART = FALSE
  LDAT_ACT = LCPDAT2
  FDAT_ACT = FP4
  BAS(#CP_PARAMS, gArcBasVelDefinition)
  SET_CD_PARAMS (0)
  TRIGGER WHEN PATH = ArcGetPath(#ArcOffBefore, WDAT2) DELAY = 0 DO ArcMainNG(#ArcOffBeforeOffStd, WDAT2, WP4) PRIO = -1
  TRIGGER WHEN PATH = ArcGetPath(#OnTheFlyArcOff, WDAT2) DELAY = 0 DO ArcMainNG(#ArcOffMoveStd, WDAT2, WP4) PRIO = -1
  ArcMainNG(#ArcOffBeforeMoveStd, WDAT2, WP4)
  LIN XP4
  ArcMainNG(#ArcOffAfterMoveStd, WDAT2, WP4)
;ENDFOLD
   $VEL.CP = 0.080
   LIN  {X 4.202, Y -7.677, Z 3.100, A 0.000, B 0.000, C 0.000} C_DIS

;FOLD ARCON WDAT1 LIN P3 Vel=0.5 m/s CPDAT1 Tool[1]:cmttorch Base[1]:vrashatel ;%{PE}
  ;FOLD Parameters ;%{h}
    ;Params IlfProvider=kukaroboter.arctech.arconlin; Kuka.IsGlobalPoint=False; Kuka.PointName=P3; Kuka.BlendingEnabled=False; Kuka.MoveDataName=CPDAT1; Kuka.VelocityPath=0.5; Kuka.CurrentCDSetIndex=0; Kuka.MovementParameterFieldEnabled=True; ArcTech.WdatVarName=WDAT1; ArcTech.Basic=3.4.3.1264
  ;ENDFOLD
  $BWDSTART = FALSE
  LDAT_ACT = LCPDAT1
  FDAT_ACT = FP3
  BAS(#CP_PARAMS, 0.5)
  SET_CD_PARAMS (0)
  TRIGGER WHEN DISTANCE = 1 DELAY = ArcGetDelay(#PreDefinition, WDAT1) DO ArcMainNG(#PreDefinition, WDAT1, WP3) PRIO = -1
  TRIGGER WHEN PATH = ArcGetPath(#OnTheFlyArcOn, WDAT1) DELAY = ArcGetDelay(#GasPreflow, WDAT1) DO ArcMainNG(#GasPreflow, WDAT1, WP3) PRIO = -1
  TRIGGER WHEN PATH = ArcGetPath(#OnTheFlyArcOn, WDAT1) DELAY = 0 DO ArcMainNG(#ArcOnMoveStd, WDAT1, WP3) PRIO = -1
  ArcMainNG(#ArcOnBeforeMoveStd, WDAT1, WP3)
  LIN XP3
  ArcMainNG(#ArcOnAfterMoveStd, WDAT1, WP3)
;ENDFOLD
   $VEL.CP = 0.060
   LIN  {X 3.050, Y -8.828, Z 3.100, A 0.000, B 0.000, C 0.000} C_DIS

;FOLD ARCOFF WDAT2 LIN P4 CPDAT2 Tool[1]:cmttorch Base[1]:vrashatel ;%{PE}
  ;FOLD Parameters ;%{h}
    ;Params IlfProvider=kukaroboter.arctech.arcofflin; Kuka.IsGlobalPoint=False; Kuka.PointName=P4; Kuka.BlendingEnabled=False; Kuka.MoveDataName=CPDAT2; Kuka.VelocityPath=0.01; Kuka.CurrentCDSetIndex=0; Kuka.MovementParameterFieldEnabled=True; ArcTech.WdatVarName=WDAT2; ArcTech.Basic=3.4.3.1264
  ;ENDFOLD
  $BWDSTART = FALSE
  LDAT_ACT = LCPDAT2
  FDAT_ACT = FP4
  BAS(#CP_PARAMS, gArcBasVelDefinition)
  SET_CD_PARAMS (0)
  TRIGGER WHEN PATH = ArcGetPath(#ArcOffBefore, WDAT2) DELAY = 0 DO ArcMainNG(#ArcOffBeforeOffStd, WDAT2, WP4) PRIO = -1
  TRIGGER WHEN PATH = ArcGetPath(#OnTheFlyArcOff, WDAT2) DELAY = 0 DO ArcMainNG(#ArcOffMoveStd, WDAT2, WP4) PRIO = -1
  ArcMainNG(#ArcOffBeforeMoveStd, WDAT2, WP4)
  LIN XP4
  ArcMainNG(#ArcOffAfterMoveStd, WDAT2, WP4)
;ENDFOLD
   $VEL.CP = 0.080
   LIN  {X 3.616, Y -8.828, Z 3.100, A 0.000, B 0.000, C 0.000} C_DIS

;FOLD ARCON WDAT1 LIN P3 Vel=0.5 m/s CPDAT1 Tool[1]:cmttorch Base[1]:vrashatel ;%{PE}
  ;FOLD Parameters ;%{h}
    ;Params IlfProvider=kukaroboter.arctech.arconlin; Kuka.IsGlobalPoint=False; Kuka.PointName=P3; Kuka.BlendingEnabled=False; Kuka.MoveDataName=CPDAT1; Kuka.VelocityPath=0.5; Kuka.CurrentCDSetIndex=0; Kuka.MovementParameterFieldEnabled=True; ArcTech.WdatVarName=WDAT1; ArcTech.Basic=3.4.3.1264
  ;ENDFOLD
  $BWDSTART = FALSE
  LDAT_ACT = LCPDAT1
  FDAT_ACT = FP3
  BAS(#CP_PARAMS, 0.5)
  SET_CD_PARAMS (0)
  TRIGGER WHEN DISTANCE = 1 DELAY = ArcGetDelay(#PreDefinition, WDAT1) DO ArcMainNG(#PreDefinition, WDAT1, WP3) PRIO = -1
  TRIGGER WHEN PATH = ArcGetPath(#OnTheFlyArcOn, WDAT1) DELAY = ArcGetDelay(#GasPreflow, WDAT1) DO ArcMainNG(#GasPreflow, WDAT1, WP3) PRIO = -1
  TRIGGER WHEN PATH = ArcGetPath(#OnTheFlyArcOn, WDAT1) DELAY = 0 DO ArcMainNG(#ArcOnMoveStd, WDAT1, WP3) PRIO = -1
  ArcMainNG(#ArcOnBeforeMoveStd, WDAT1, WP3)
  LIN XP3
  ArcMainNG(#ArcOnAfterMoveStd, WDAT1, WP3)
;ENDFOLD
   $VEL.CP = 0.060
   LIN  {X 4.668, Y -7.776, Z 3.100, A 0.000, B 0.000, C 0.000} C_DIS

;FOLD ARCOFF WDAT2 LIN P4 CPDAT2 Tool[1]:cmttorch Base[1]:vrashatel ;%{PE}
  ;FOLD Parameters ;%{h}
    ;Params IlfProvider=kukaroboter.arctech.arcofflin; Kuka.IsGlobalPoint=False; Kuka.PointName=P4; Kuka.BlendingEnabled=False; Kuka.MoveDataName=CPDAT2; Kuka.VelocityPath=0.01; Kuka.CurrentCDSetIndex=0; Kuka.MovementParameterFieldEnabled=True; ArcTech.WdatVarName=WDAT2; ArcTech.Basic=3.4.3.1264
  ;ENDFOLD
  $BWDSTART = FALSE
  LDAT_ACT = LCPDAT2
  FDAT_ACT = FP4
  BAS(#CP_PARAMS, gArcBasVelDefinition)
  SET_CD_PARAMS (0)
  TRIGGER WHEN PATH = ArcGetPath(#ArcOffBefore, WDAT2) DELAY = 0 DO ArcMainNG(#ArcOffBeforeOffStd, WDAT2, WP4) PRIO = -1
  TRIGGER WHEN PATH = ArcGetPath(#OnTheFlyArcOff, WDAT2) DELAY = 0 DO ArcMainNG(#ArcOffMoveStd, WDAT2, WP4) PRIO = -1
  ArcMainNG(#ArcOffBeforeMoveStd, WDAT2, WP4)
  LIN XP4
  ArcMainNG(#ArcOffAfterMoveStd, WDAT2, WP4)
;ENDFOLD
   $VEL.CP = 0.080
   LIN  {X 4.669, Y -8.341, Z 3.100, A 0.000, B 0.000, C 0.000} C_DIS

;FOLD ARCON WDAT1 LIN P3 Vel=0.5 m/s CPDAT1 Tool[1]:cmttorch Base[1]:vrashatel ;%{PE}
  ;FOLD Parameters ;%{h}
    ;Params IlfProvider=kukaroboter.arctech.arconlin; Kuka.IsGlobalPoint=False; Kuka.PointName=P3; Kuka.BlendingEnabled=False; Kuka.MoveDataName=CPDAT1; Kuka.VelocityPath=0.5; Kuka.CurrentCDSetIndex=0; Kuka.MovementParameterFieldEnabled=True; ArcTech.WdatVarName=WDAT1; ArcTech.Basic=3.4.3.1264
  ;ENDFOLD
  $BWDSTART = FALSE
  LDAT_ACT = LCPDAT1
  FDAT_ACT = FP3
  BAS(#CP_PARAMS, 0.5)
  SET_CD_PARAMS (0)
  TRIGGER WHEN DISTANCE = 1 DELAY = ArcGetDelay(#PreDefinition, WDAT1) DO ArcMainNG(#PreDefinition, WDAT1, WP3) PRIO = -1
  TRIGGER WHEN PATH = ArcGetPath(#OnTheFlyArcOn, WDAT1) DELAY = ArcGetDelay(#GasPreflow, WDAT1) DO ArcMainNG(#GasPreflow, WDAT1, WP3) PRIO = -1
  TRIGGER WHEN PATH = ArcGetPath(#OnTheFlyArcOn, WDAT1) DELAY = 0 DO ArcMainNG(#ArcOnMoveStd, WDAT1, WP3) PRIO = -1
  ArcMainNG(#ArcOnBeforeMoveStd, WDAT1, WP3)
  LIN XP3
  ArcMainNG(#ArcOnAfterMoveStd, WDAT1, WP3)
;ENDFOLD
   $VEL.CP = 0.060
   LIN  {X 4.181, Y -8.828, Z 3.100, A 0.000, B 0.000, C 0.000} C_DIS

;FOLD ARCOFF WDAT2 LIN P4 CPDAT2 Tool[1]:cmttorch Base[1]:vrashatel ;%{PE}
  ;FOLD Parameters ;%{h}
    ;Params IlfProvider=kukaroboter.arctech.arcofflin; Kuka.IsGlobalPoint=False; Kuka.PointName=P4; Kuka.BlendingEnabled=False; Kuka.MoveDataName=CPDAT2; Kuka.VelocityPath=0.01; Kuka.CurrentCDSetIndex=0; Kuka.MovementParameterFieldEnabled=True; ArcTech.WdatVarName=WDAT2; ArcTech.Basic=3.4.3.1264
  ;ENDFOLD
  $BWDSTART = FALSE
  LDAT_ACT = LCPDAT2
  FDAT_ACT = FP4
  BAS(#CP_PARAMS, gArcBasVelDefinition)
  SET_CD_PARAMS (0)
  TRIGGER WHEN PATH = ArcGetPath(#ArcOffBefore, WDAT2) DELAY = 0 DO ArcMainNG(#ArcOffBeforeOffStd, WDAT2, WP4) PRIO = -1
  TRIGGER WHEN PATH = ArcGetPath(#OnTheFlyArcOff, WDAT2) DELAY = 0 DO ArcMainNG(#ArcOffMoveStd, WDAT2, WP4) PRIO = -1
  ArcMainNG(#ArcOffBeforeMoveStd, WDAT2, WP4)
  LIN XP4
  ArcMainNG(#ArcOffAfterMoveStd, WDAT2, WP4)
;ENDFOLD
   $VEL.CP = 0.080
   LIN  {X 4.181, Y -9.290, Z 3.100, A 0.000, B 0.000, C 0.000} C_DIS
   $VEL.CP = 0.080
   LIN  {X 4.868, Y -9.218, Z 3.100, A 0.000, B 0.000, C 0.000} C_DIS
   $VEL.CP = 0.080
   LIN  {X 7.385, Y -1.843, Z 3.100, A 0.000, B 0.000, C 0.000} C_DIS
   $VEL.CP = 0.080
   LIN  {X 7.445, Y -1.783, Z 3.100, A 0.000, B 0.000, C 0.000} C_DIS

;FOLD ARCON WDAT1 LIN P3 Vel=0.5 m/s CPDAT1 Tool[1]:cmttorch Base[1]:vrashatel ;%{PE}
  ;FOLD Parameters ;%{h}
    ;Params IlfProvider=kukaroboter.arctech.arconlin; Kuka.IsGlobalPoint=False; Kuka.PointName=P3; Kuka.BlendingEnabled=False; Kuka.MoveDataName=CPDAT1; Kuka.VelocityPath=0.5; Kuka.CurrentCDSetIndex=0; Kuka.MovementParameterFieldEnabled=True; ArcTech.WdatVarName=WDAT1; ArcTech.Basic=3.4.3.1264
  ;ENDFOLD
  $BWDSTART = FALSE
  LDAT_ACT = LCPDAT1
  FDAT_ACT = FP3
  BAS(#CP_PARAMS, 0.5)
  SET_CD_PARAMS (0)
  TRIGGER WHEN DISTANCE = 1 DELAY = ArcGetDelay(#PreDefinition, WDAT1) DO ArcMainNG(#PreDefinition, WDAT1, WP3) PRIO = -1
  TRIGGER WHEN PATH = ArcGetPath(#OnTheFlyArcOn, WDAT1) DELAY = ArcGetDelay(#GasPreflow, WDAT1) DO ArcMainNG(#GasPreflow, WDAT1, WP3) PRIO = -1
  TRIGGER WHEN PATH = ArcGetPath(#OnTheFlyArcOn, WDAT1) DELAY = 0 DO ArcMainNG(#ArcOnMoveStd, WDAT1, WP3) PRIO = -1
  ArcMainNG(#ArcOnBeforeMoveStd, WDAT1, WP3)
  LIN XP3
  ArcMainNG(#ArcOnAfterMoveStd, WDAT1, WP3)
;ENDFOLD
   $VEL.CP = 0.060
   LIN  {X 9.010, Y -1.783, Z 3.100, A 0.000, B 0.000, C 0.000} C_DIS
   $VEL.CP = 0.060
   LIN  {X 9.010, Y 1.118, Z 3.100, A 0.000, B 0.000, C 0.000} C_DIS
   $VEL.CP = 0.060
   LIN  {X 7.445, Y 1.118, Z 3.100, A 0.000, B 0.000, C 0.000} C_DIS
   $VEL.CP = 0.060
   LIN  {X 7.445, Y -1.783, Z 3.100, A 0.000, B 0.000, C 0.000} C_DIS

;FOLD ARCOFF WDAT2 LIN P4 CPDAT2 Tool[1]:cmttorch Base[1]:vrashatel ;%{PE}
  ;FOLD Parameters ;%{h}
    ;Params IlfProvider=kukaroboter.arctech.arcofflin; Kuka.IsGlobalPoint=False; Kuka.PointName=P4; Kuka.BlendingEnabled=False; Kuka.MoveDataName=CPDAT2; Kuka.VelocityPath=0.01; Kuka.CurrentCDSetIndex=0; Kuka.MovementParameterFieldEnabled=True; ArcTech.WdatVarName=WDAT2; ArcTech.Basic=3.4.3.1264
  ;ENDFOLD
  $BWDSTART = FALSE
  LDAT_ACT = LCPDAT2
  FDAT_ACT = FP4
  BAS(#CP_PARAMS, gArcBasVelDefinition)
  SET_CD_PARAMS (0)
  TRIGGER WHEN PATH = ArcGetPath(#ArcOffBefore, WDAT2) DELAY = 0 DO ArcMainNG(#ArcOffBeforeOffStd, WDAT2, WP4) PRIO = -1
  TRIGGER WHEN PATH = ArcGetPath(#OnTheFlyArcOff, WDAT2) DELAY = 0 DO ArcMainNG(#ArcOffMoveStd, WDAT2, WP4) PRIO = -1
  ArcMainNG(#ArcOffBeforeMoveStd, WDAT2, WP4)
  LIN XP4
  ArcMainNG(#ArcOffAfterMoveStd, WDAT2, WP4)
;ENDFOLD
   $VEL.CP = 0.080
   LIN  {X 7.385, Y -1.843, Z 3.100, A 0.000, B 0.000, C 0.000} C_DIS
   $VEL.CP = 0.080
   LIN  {X 9.218, Y -1.801, Z 3.100, A 0.000, B 0.000, C 0.000} C_DIS
   $VEL.CP = 0.080
   LIN  {X 9.290, Y -1.352, Z 3.100, A 0.000, B 0.000, C 0.000} C_DIS
   $VEL.CP = 0.080
   LIN  {X 8.829, Y -1.352, Z 3.100, A 0.000, B 0.000, C 0.000} C_DIS

;FOLD ARCON WDAT1 LIN P3 Vel=0.5 m/s CPDAT1 Tool[1]:cmttorch Base[1]:vrashatel ;%{PE}
  ;FOLD Parameters ;%{h}
    ;Params IlfProvider=kukaroboter.arctech.arconlin; Kuka.IsGlobalPoint=False; Kuka.PointName=P3; Kuka.BlendingEnabled=False; Kuka.MoveDataName=CPDAT1; Kuka.VelocityPath=0.5; Kuka.CurrentCDSetIndex=0; Kuka.MovementParameterFieldEnabled=True; ArcTech.WdatVarName=WDAT1; ArcTech.Basic=3.4.3.1264
  ;ENDFOLD
  $BWDSTART = FALSE
  LDAT_ACT = LCPDAT1
  FDAT_ACT = FP3
  BAS(#CP_PARAMS, 0.5)
  SET_CD_PARAMS (0)
  TRIGGER WHEN DISTANCE = 1 DELAY = ArcGetDelay(#PreDefinition, WDAT1) DO ArcMainNG(#PreDefinition, WDAT1, WP3) PRIO = -1
  TRIGGER WHEN PATH = ArcGetPath(#OnTheFlyArcOn, WDAT1) DELAY = ArcGetDelay(#GasPreflow, WDAT1) DO ArcMainNG(#GasPreflow, WDAT1, WP3) PRIO = -1
  TRIGGER WHEN PATH = ArcGetPath(#OnTheFlyArcOn, WDAT1) DELAY = 0 DO ArcMainNG(#ArcOnMoveStd, WDAT1, WP3) PRIO = -1
  ArcMainNG(#ArcOnBeforeMoveStd, WDAT1, WP3)
  LIN XP3
  ArcMainNG(#ArcOnAfterMoveStd, WDAT1, WP3)
;ENDFOLD
   $VEL.CP = 0.060
   LIN  {X 8.579, Y -1.603, Z 3.100, A 0.000, B 0.000, C 0.000} C_DIS

;FOLD ARCOFF WDAT2 LIN P4 CPDAT2 Tool[1]:cmttorch Base[1]:vrashatel ;%{PE}
  ;FOLD Parameters ;%{h}
    ;Params IlfProvider=kukaroboter.arctech.arcofflin; Kuka.IsGlobalPoint=False; Kuka.PointName=P4; Kuka.BlendingEnabled=False; Kuka.MoveDataName=CPDAT2; Kuka.VelocityPath=0.01; Kuka.CurrentCDSetIndex=0; Kuka.MovementParameterFieldEnabled=True; ArcTech.WdatVarName=WDAT2; ArcTech.Basic=3.4.3.1264
  ;ENDFOLD
  $BWDSTART = FALSE
  LDAT_ACT = LCPDAT2
  FDAT_ACT = FP4
  BAS(#CP_PARAMS, gArcBasVelDefinition)
  SET_CD_PARAMS (0)
  TRIGGER WHEN PATH = ArcGetPath(#ArcOffBefore, WDAT2) DELAY = 0 DO ArcMainNG(#ArcOffBeforeOffStd, WDAT2, WP4) PRIO = -1
  TRIGGER WHEN PATH = ArcGetPath(#OnTheFlyArcOff, WDAT2) DELAY = 0 DO ArcMainNG(#ArcOffMoveStd, WDAT2, WP4) PRIO = -1
  ArcMainNG(#ArcOffBeforeMoveStd, WDAT2, WP4)
  LIN XP4
  ArcMainNG(#ArcOffAfterMoveStd, WDAT2, WP4)
;ENDFOLD
   $VEL.CP = 0.080
   LIN  {X 8.013, Y -1.603, Z 3.100, A 0.000, B 0.000, C 0.000} C_DIS

;FOLD ARCON WDAT1 LIN P3 Vel=0.5 m/s CPDAT1 Tool[1]:cmttorch Base[1]:vrashatel ;%{PE}
  ;FOLD Parameters ;%{h}
    ;Params IlfProvider=kukaroboter.arctech.arconlin; Kuka.IsGlobalPoint=False; Kuka.PointName=P3; Kuka.BlendingEnabled=False; Kuka.MoveDataName=CPDAT1; Kuka.VelocityPath=0.5; Kuka.CurrentCDSetIndex=0; Kuka.MovementParameterFieldEnabled=True; ArcTech.WdatVarName=WDAT1; ArcTech.Basic=3.4.3.1264
  ;ENDFOLD
  $BWDSTART = FALSE
  LDAT_ACT = LCPDAT1
  FDAT_ACT = FP3
  BAS(#CP_PARAMS, 0.5)
  SET_CD_PARAMS (0)
  TRIGGER WHEN DISTANCE = 1 DELAY = ArcGetDelay(#PreDefinition, WDAT1) DO ArcMainNG(#PreDefinition, WDAT1, WP3) PRIO = -1
  TRIGGER WHEN PATH = ArcGetPath(#OnTheFlyArcOn, WDAT1) DELAY = ArcGetDelay(#GasPreflow, WDAT1) DO ArcMainNG(#GasPreflow, WDAT1, WP3) PRIO = -1
  TRIGGER WHEN PATH = ArcGetPath(#OnTheFlyArcOn, WDAT1) DELAY = 0 DO ArcMainNG(#ArcOnMoveStd, WDAT1, WP3) PRIO = -1
  ArcMainNG(#ArcOnBeforeMoveStd, WDAT1, WP3)
  LIN XP3
  ArcMainNG(#ArcOnAfterMoveStd, WDAT1, WP3)
;ENDFOLD
   $VEL.CP = 0.060
   LIN  {X 8.829, Y -0.787, Z 3.100, A 0.000, B 0.000, C 0.000} C_DIS

;FOLD ARCOFF WDAT2 LIN P4 CPDAT2 Tool[1]:cmttorch Base[1]:vrashatel ;%{PE}
  ;FOLD Parameters ;%{h}
    ;Params IlfProvider=kukaroboter.arctech.arcofflin; Kuka.IsGlobalPoint=False; Kuka.PointName=P4; Kuka.BlendingEnabled=False; Kuka.MoveDataName=CPDAT2; Kuka.VelocityPath=0.01; Kuka.CurrentCDSetIndex=0; Kuka.MovementParameterFieldEnabled=True; ArcTech.WdatVarName=WDAT2; ArcTech.Basic=3.4.3.1264
  ;ENDFOLD
  $BWDSTART = FALSE
  LDAT_ACT = LCPDAT2
  FDAT_ACT = FP4
  BAS(#CP_PARAMS, gArcBasVelDefinition)
  SET_CD_PARAMS (0)
  TRIGGER WHEN PATH = ArcGetPath(#ArcOffBefore, WDAT2) DELAY = 0 DO ArcMainNG(#ArcOffBeforeOffStd, WDAT2, WP4) PRIO = -1
  TRIGGER WHEN PATH = ArcGetPath(#OnTheFlyArcOff, WDAT2) DELAY = 0 DO ArcMainNG(#ArcOffMoveStd, WDAT2, WP4) PRIO = -1
  ArcMainNG(#ArcOffBeforeMoveStd, WDAT2, WP4)
  LIN XP4
  ArcMainNG(#ArcOffAfterMoveStd, WDAT2, WP4)
;ENDFOLD
   $VEL.CP = 0.080
   LIN  {X 8.829, Y -0.221, Z 3.100, A 0.000, B 0.000, C 0.000} C_DIS

;FOLD ARCON WDAT1 LIN P3 Vel=0.5 m/s CPDAT1 Tool[1]:cmttorch Base[1]:vrashatel ;%{PE}
  ;FOLD Parameters ;%{h}
    ;Params IlfProvider=kukaroboter.arctech.arconlin; Kuka.IsGlobalPoint=False; Kuka.PointName=P3; Kuka.BlendingEnabled=False; Kuka.MoveDataName=CPDAT1; Kuka.VelocityPath=0.5; Kuka.CurrentCDSetIndex=0; Kuka.MovementParameterFieldEnabled=True; ArcTech.WdatVarName=WDAT1; ArcTech.Basic=3.4.3.1264
  ;ENDFOLD
  $BWDSTART = FALSE
  LDAT_ACT = LCPDAT1
  FDAT_ACT = FP3
  BAS(#CP_PARAMS, 0.5)
  SET_CD_PARAMS (0)
  TRIGGER WHEN DISTANCE = 1 DELAY = ArcGetDelay(#PreDefinition, WDAT1) DO ArcMainNG(#PreDefinition, WDAT1, WP3) PRIO = -1
  TRIGGER WHEN PATH = ArcGetPath(#OnTheFlyArcOn, WDAT1) DELAY = ArcGetDelay(#GasPreflow, WDAT1) DO ArcMainNG(#GasPreflow, WDAT1, WP3) PRIO = -1
  TRIGGER WHEN PATH = ArcGetPath(#OnTheFlyArcOn, WDAT1) DELAY = 0 DO ArcMainNG(#ArcOnMoveStd, WDAT1, WP3) PRIO = -1
  ArcMainNG(#ArcOnBeforeMoveStd, WDAT1, WP3)
  LIN XP3
  ArcMainNG(#ArcOnAfterMoveStd, WDAT1, WP3)
;ENDFOLD
   $VEL.CP = 0.060
   LIN  {X 7.624, Y -1.426, Z 3.100, A 0.000, B 0.000, C 0.000} C_DIS

;FOLD ARCOFF WDAT2 LIN P4 CPDAT2 Tool[1]:cmttorch Base[1]:vrashatel ;%{PE}
  ;FOLD Parameters ;%{h}
    ;Params IlfProvider=kukaroboter.arctech.arcofflin; Kuka.IsGlobalPoint=False; Kuka.PointName=P4; Kuka.BlendingEnabled=False; Kuka.MoveDataName=CPDAT2; Kuka.VelocityPath=0.01; Kuka.CurrentCDSetIndex=0; Kuka.MovementParameterFieldEnabled=True; ArcTech.WdatVarName=WDAT2; ArcTech.Basic=3.4.3.1264
  ;ENDFOLD
  $BWDSTART = FALSE
  LDAT_ACT = LCPDAT2
  FDAT_ACT = FP4
  BAS(#CP_PARAMS, gArcBasVelDefinition)
  SET_CD_PARAMS (0)
  TRIGGER WHEN PATH = ArcGetPath(#ArcOffBefore, WDAT2) DELAY = 0 DO ArcMainNG(#ArcOffBeforeOffStd, WDAT2, WP4) PRIO = -1
  TRIGGER WHEN PATH = ArcGetPath(#OnTheFlyArcOff, WDAT2) DELAY = 0 DO ArcMainNG(#ArcOffMoveStd, WDAT2, WP4) PRIO = -1
  ArcMainNG(#ArcOffBeforeMoveStd, WDAT2, WP4)
  LIN XP4
  ArcMainNG(#ArcOffAfterMoveStd, WDAT2, WP4)
;ENDFOLD
   $VEL.CP = 0.080
   LIN  {X 7.624, Y -0.861, Z 3.100, A 0.000, B 0.000, C 0.000} C_DIS

;FOLD ARCON WDAT1 LIN P3 Vel=0.5 m/s CPDAT1 Tool[1]:cmttorch Base[1]:vrashatel ;%{PE}
  ;FOLD Parameters ;%{h}
    ;Params IlfProvider=kukaroboter.arctech.arconlin; Kuka.IsGlobalPoint=False; Kuka.PointName=P3; Kuka.BlendingEnabled=False; Kuka.MoveDataName=CPDAT1; Kuka.VelocityPath=0.5; Kuka.CurrentCDSetIndex=0; Kuka.MovementParameterFieldEnabled=True; ArcTech.WdatVarName=WDAT1; ArcTech.Basic=3.4.3.1264
  ;ENDFOLD
  $BWDSTART = FALSE
  LDAT_ACT = LCPDAT1
  FDAT_ACT = FP3
  BAS(#CP_PARAMS, 0.5)
  SET_CD_PARAMS (0)
  TRIGGER WHEN DISTANCE = 1 DELAY = ArcGetDelay(#PreDefinition, WDAT1) DO ArcMainNG(#PreDefinition, WDAT1, WP3) PRIO = -1
  TRIGGER WHEN PATH = ArcGetPath(#OnTheFlyArcOn, WDAT1) DELAY = ArcGetDelay(#GasPreflow, WDAT1) DO ArcMainNG(#GasPreflow, WDAT1, WP3) PRIO = -1
  TRIGGER WHEN PATH = ArcGetPath(#OnTheFlyArcOn, WDAT1) DELAY = 0 DO ArcMainNG(#ArcOnMoveStd, WDAT1, WP3) PRIO = -1
  ArcMainNG(#ArcOnBeforeMoveStd, WDAT1, WP3)
  LIN XP3
  ArcMainNG(#ArcOnAfterMoveStd, WDAT1, WP3)
;ENDFOLD
   $VEL.CP = 0.060
   LIN  {X 8.829, Y 0.344, Z 3.100, A 0.000, B 0.000, C 0.000} C_DIS

